# B&R Automation Studio project PrintMark
Automation Studio 4.12.2.93; technology packages: Acp10Arnc0 5.24.1, mapp 5.24.2, mappView 5.24.1

## Configuration Config1

CPU X20CP1584, AutomationRuntime B4.93, Build 4.1.2, Vc V4.72.6

### Task classes (Cpu.sw)
```
Cyclic#1 (cycle 1600 us, tolerance 1600 us):
  BeltCtrl <- SOURCE.BeltCtrl.BeltCtrl.prg  // This task is for controlling the belt conveyor
  CutterCtrl <- SOURCE.CutterCtrl.CutterCtrl.prg  // This task is for controlling the cutter axis
  RegMkCtrl <- SOURCE.RegMark.RegMkCtrl.prg  // This task is for reg mark capture
Cyclic#4 (cycle 99200 us, tolerance 99200 us):
  VisCtrl <- SOURCE.VisCtrl.VisCtrl.prg  // This task if for Hmi task control
  MainCtrl <- SOURCE.MainCtrl.MainCtrl.prg
DataObjects: Acp10sys
NcDataObjects: acp10etxen <- acp10etxen.dob, gBeltAxisa <- gBeltAxisobj.gBeltAxisa.dob, gBeltAxisi <- gBeltAxisobj.gBeltAxisi.dob, gCutAxisa <- gCutAxisobj.gCutAxisa.dob, gCutAxisi <- gCutAxisobj.gCutAxisi.dob
Binaries: FWRules, TCData, udbdef, TCLang, arsvcreg, mvLoader, acp10cfg, Acp10map, iomap, arconfig, asfw, ashwac, sysconf, User, Role, ashwd, BeltConfig, TC, CutConfig, PrintAlarm, PrintCom
Libraries: Acp10man, Acp10par, NcGlobal, Acp10_MC, sys_lib, brsystem, runtime, MpPackML, MpBase, astime, MpAxis, MpCom, standard, MpAlarmX, MpServer, MC_RegMa, fileio, powerlnk, arssl, asbrstr, asieccon, dataobj, aruser
```

### Hardware
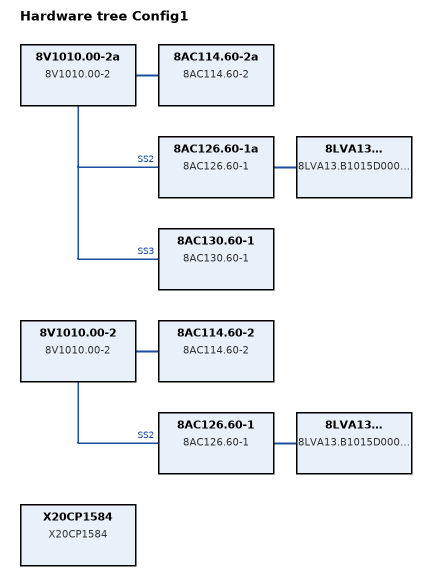
```
8AC114.60-2 : 8AC114.60-2 v1.0.0.8  [SS -> 8V1010.00-2.SS1; PLK1 -> X20CP1584.IF3 (NodeNumber=1) [Cable Type=PowerlinkCable, Length=10, Version=1.0.0.3]; PLK2 -> 8AC114.60-2a.PLK1 (NodeNumber=1) [Cable Type=PowerlinkCable, Length=10, Version=1.0.0.3]]
8AC114.60-2a : 8AC114.60-2 v1.0.0.8  [SS -> 8V1010.00-2a.SS1; PLK1 -> 8AC114.60-2.PLK2 (NodeNumber=2) [Cable Type=PowerlinkCable, Length=10, Version=1.0.0.3]]
8AC126.60-1 : 8AC126.60-1 v2.2.0.0  [SS -> 8V1010.00-2.SS2]
8AC126.60-1a : 8AC126.60-1 v2.2.0.0  [SS -> 8V1010.00-2a.SS2]
8AC130.60-1 : 8AC130.60-1 v2.2.0.0  [SS -> 8V1010.00-2a.SS3]
8LVA13.B1015D000-0 : 8LVA13.B1015D000-0 v2.2.0.3  [EC -> 8AC126.60-1.EC; MT -> 8V1010.00-2.MT1]
8LVA13.B1015D000-0a : 8LVA13.B1015D000-0 v2.2.0.3  [EC -> 8AC126.60-1a.EC; MT -> 8V1010.00-2a.MT1]
8V1010.00-2 : 8V1010.00-2 v2.2.0.0
  MotionTP = Acp10Arnc0
  SinglePhaseOperation = on
  BothEndSwitchesAreNormallyOpen_r1 = on
  QuickStopIsNormallyOpen_r1 = on
8V1010.00-2a : 8V1010.00-2 v2.2.0.0
  MotionTP = Acp10Arnc0
  SinglePhaseOperation = on
  AxisIsPeriodic_r1 = on
  Period_r1 = 3600
  BothEndSwitchesAreNormallyOpen_r1 = on
  QuickStopIsNormallyOpen_r1 = on
X20CP1584 : X20CP1584 v1.10.0.0
  Connector IF2:
    ActivateDevice = 1
    Mode = Manual
    InternetAddress = 192.168.0.11
    SubnetMask = 255.255.255.0
    ActivateSnmp = 2
  Connector IF3:
    CycleTime = 1600
  ConfigurationID = PrintMark_Config1
  TimerDeviceType = EPLX2X
  TimerDevice = X20CP1584.IF3
  TaskClassIdleTime = 1600
  Cyclic1Duration = 1600
  Cyclic1Tolerance = 1600
  Cyclic2Duration = 19200
  Cyclic2Tolerance = 19200
  Cyclic3Duration = 49600
  Cyclic3Tolerance = 49600
  Cyclic4Duration = 99200
  Cyclic4Tolerance = 99200
  Cyclic6Duration = 499200
  Cyclic6Tolerance = 499200
  Cyclic8Duration = 9600
  FileDevice1
  FileDeviceName1 = USER
  FileDevicePath1 = USER_PATH
  FileDevice2
  FileDeviceName2 = Print
  FileDevicePath2 = C:\
  FtpUser1
  FtpUsername1 = printmark
  FtpUserPassword1 = J40jtcY6ygfeMe3/XVHLOVhutVx6SKtWgX0BANt4QHs=
  FtpUserSalt1 = 8YC+oSMn
  FTPAccessRight1 = 0
  FTPdevice1 = ALL
  ActivateOpcUa = 1
  OpcUaInformationModels_PV_Version = 1
```

### Acp10cfg.ncc - X20CP1584/Motion/Acp10cfg.ncc
```
NcConfiguration (Version=5.24.1, NcSwId=Acp10)
  ACP10CF1_typ:
    cnt_nettrc_rec_drive = 1500
    bufsize_trace_upload = 1200
    tc_nc_man_task = Cyclic #1
    glob_pv_as_ncobject = Yes
    ncsys_dl_broadcast = Yes
    ncsys_dl_acp_reset = Yes
    safemc_log_err_to_ax = Yes
    network_init:
      ncsw_init_execute = Yes
      automatic_execute = Yes
      node_nr_warning = Yes
      net_err_before_ncact = Yes
    nettrc:
      enter_parsecrec = Yes
      enter_ncaction = Yes
      save_ring_startidx = Yes
    cam_prof_download:
      cam_dat_dl_parallel = No
      tc_cam_dl_parallel = Task class for NC Manager task
    plk_if[0]:
      if_name = IF3
      tc_CycDat_PLCopen = Task class for NC Manager task
      mc_broadcast_extdat = No
```

### Acp10map.ncm - X20CP1584/Motion/Acp10map.ncm
```
NcMapping (NcSwId=Acp10, DisabledNodesAreHidden=False)
  NcObject 8V1010.00-2_ncV_AXIS1 (ModuleId=8V1010.00-2, Type=ncV_AXIS, Channel=1, Disabled=TRUE, ModuleDisabled=FALSE)
  NcObject 8V1010.00-2a_ncV_AXIS1 (ModuleId=8V1010.00-2a, Type=ncV_AXIS, Channel=1, Disabled=TRUE, ModuleDisabled=FALSE)
  NcObject gBeltAxis (ModuleId=8V1010.00-2, Type=ncAXIS, Channel=1, AcoposSimulation=Off, InitParameter=gBeltAxisi, AcoposParameter=gBeltAxisa, Disabled=FALSE, ModuleDisabled=FALSE)  // This axis is for Belt conveyor
  NcObject gCutAxis (ModuleId=8V1010.00-2a, Type=ncAXIS, Channel=1, AcoposSimulation=Off, InitParameter=gCutAxisi, AcoposParameter=gCutAxisa, AdditionalData=PLCopen_ModPos="3600,1" , Disabled=FALSE, ModuleDisabled=FALSE)  // This axis is for Cutter unit
```

### BeltConfig.mpaxisbasic - X20CP1584/Motion/BeltConfig.mpaxisbasic
```
Element gMl_BeltAxis (Type=mpaxisbasic)
  Alarms = MpAlarmX
```

### CutConfig.mpaxisbasic - X20CP1584/Motion/CutConfig.mpaxisbasic
```
Element gMl_CutAxis (Type=mpaxisbasic)
  Alarms = MpAlarmX
```

### PrintAlarm.mpalarmxcore - X20CP1584/mappServices/PrintAlarm.mpalarmxcore
```
Element gMl_PrintAlarm (Type=mpalarmxcore)
  mapp.AlarmX.Core.Configuration:
    [0]:
      Name = Estop
      Message = Machine E-Stop is pressed
      Behavior = PersistentAlarm
    [1]:
      Name = BeltTempError
      Message = Belt conveyor motor temperature is high
      Behavior = PersistentAlarm
    [2]:
      Name = CutterTempError
      Message = Cutter conveyor motor is temperature is high
      Behavior = PersistentAlarm
    [3]:
      Name = CuttingZone
      Message = Cutter is in cutting zone please move it manually
      Behavior = PersistentAlarm
```

### PrintCom.mpcomgroup - X20CP1584/mappServices/PrintCom.mpcomgroup
```
Element gMl_PrintChildGroup (Type=mpcomgroup)
  Linking:
    Subnodes:
      0 = gMl_BeltAxis
      1 = gMl_CutAxis
      2 = gMl_PrintAlarm
  Alarms = MpAlarmX
Element gMl_PrintParentGroup (Type=mpcomgroup)
  Linking:
    Subnodes:
      0 = gMl_PrintChildGroup
  Alarms = MpAlarmX
```

### PrintData.mpdatarecorder - X20CP1584/mappServices/PrintData.mpdatarecorder
```
Element gMl_PrintDataRecorder (Type=mpdatarecorder)
```

### PrintPack.mppackmlcore - X20CP1584/mappServices/PrintPack.mppackmlcore
```
Element gMl_PrintPackML (Type=mppackmlcore)
  Modes:
    Mode[1]:
      ModeID = 1
      Name = Automatic
    Mode[2]:
      ModeID = 2
      Name = Mode[3]
```

## Logical view

Binary libraries used (declarations not repeated): operator, runtime, astime, AsIecCon, Acp10man, Acp10par, NcGlobal, Acp10_MC, sys_lib, brsystem, MpPackML, MpBase, MpAxis, standard, MpAlarmX, MpServer, MC_RegMa 5.24.1

### Global.typ - Global data types
```iecst
(*Structure for axis control*)

TYPE
	AxisBasicIn_type : 	STRUCT  (*Axis Basic inputs structure type*)
		ErrorReset : BOOL; (*Resets function block errors*) (* *) (*#PAR#;*)
		Parameters : MpAxisBasicParType; (*Function block parameters*) (* *) (*#PAR#;*)
		Update : BOOL; (*Updates the parameters*) (* *) (*#PAR#;*)
		Power : BOOL; (*Level-sensitive command for turning an axis on/off. In the event of an error, a new rising edge is required to restart the axis*) (* *) (*#CMD#;*)
		Home : BOOL; (*Command for homing the axis*) (* *) (*#CMD#;*)
		MoveVelocity : BOOL; (*Starts a constant movement with a defined velocity*) (* *) (*#CMD#;*)
		MoveAbsolute : BOOL; (*Starts an absolute movement*) (* *) (*#CMD#;*)
		MoveAdditive : BOOL; (*Starts a relative movement*) (* *) (*#CMD#;*)
		Stop : BOOL; (*Stops the axis*) (* *) (*#CMD#;*)
		JogPositive : BOOL; (*Movement in the positive direction. Stops automatically at the software limit position*) (* *) (*#CMD#OPT#;*)
		JogNegative : BOOL; (*Movement in the negative direction. Stops automatically at the software limit position*) (* *) (*#CMD#OPT#;*)
		Autotune : BOOL; (*Starts autotuning*) (* *) (*#CMD#OPT#;*)
		Simulate : BOOL; (*Enables motor simulation*) (* *) (*#CMD#OPT#;*)
		TorqueLimit : BOOL; (*Enables torque limiting*) (* *) (*#CMD#OPT#;*)
		ReleaseBrake : BOOL; (*Locks or unlocks the holding brake (only when the axis is switched off)*) (* *) (*#CMD#OPT#;*)
	END_STRUCT;
	AxisBasicOut_type : 	STRUCT  (*Axis Basic outputs structure type*)
		Active : BOOL; (*Indicates whether the function block is active*) (* *) (*#PAR#;*)
		Error : BOOL; (*Indicates that the function block is in an error state or a command was not executed correctly*) (* *) (*#PAR#;*)
		StatusID : DINT; (*Status information about the function block*) (* *) (*#PAR#;*)
		UpdateDone : BOOL; (*Parameter update completed*) (* *) (*#PAR#;*)
		Position : LREAL; (*Current position of the axis [units]*) (* *) (*#CYC#;*)
		Velocity : REAL; (*Current position of the axis [units/s]*) (* *) (*#CYC#;*)
		CommandBusy : BOOL; (*Function block currently executing command*) (* *) (*#CMD#OPT#;*)
		CommandAborted : BOOL; (*Function block interrupted while executing a command*) (* *) (*#CMD#OPT#;*)
		PowerOn : BOOL; (*Switches on the axis*) (* *) (*#CMD#;*)
		IsHomed : BOOL; (*Homes the axis*) (* *) (*#CMD#;*)
		InVelocity : BOOL; (*Axis running with defined velocity*) (* *) (*#CMD#;*)
		InPosition : BOOL; (*Axis reached the desired position*) (* *) (*#CMD#;*)
		MoveActive : BOOL; (*Movement active*) (* *) (*#CMD#;*)
		Stopped : BOOL; (*Axis stopped*) (* *) (*#CMD#;*)
		TuningDone : BOOL; (*Autotuning completed successfully*) (* *) (*#CMD#OPT#;*)
		Simulation : BOOL; (*Motor simulation active*) (* *) (*#CMD#OPT#;*)
		TorqueLimited : BOOL; (*Torque limiting function active*) (* *) (*#CMD#OPT#;*)
		BrakeReleased : BOOL; (*Holding brake manually released*) (* *) (*#CMD#OPT#;*)
		Info : MpAxisBasicInfoType; (*Additional information about the component*) (* *) (*#CMD#;*)
	END_STRUCT;
	AxisBasic_type : 	STRUCT  (*Axis Basic structure type*)
		In : AxisBasicIn_type;
		Out : AxisBasicOut_type;
	END_STRUCT;
	AxisCamSeqIn_type : 	STRUCT  (*Axis cam sequencing input structure type*)
		ErrorReset : BOOL; (*Resets function block errors*) (* *) (*#PAR#;*)
		Parameters : MpAxisCamSequencerParType; (*Function block parameters*) (* *) (*#PAR#;*)
		Update : BOOL; (*Update command for the parameters*) (* *) (*#PAR#;*)
		Signal1 : BOOL; (*Sets the signal for the sequencer on a rising edge and resets the signal on a falling edge*) (* *) (*#CMD#;*)
		Signal2 : BOOL; (*Sets the signal for the sequencer on a rising edge and resets the signal on a falling edge*) (* *) (*#CMD#;*)
		Signal3 : BOOL; (*Sets the signal for the sequencer on a rising edge and resets the signal on a falling edge*) (* *) (*#CMD#OPT#;*)
		Signal4 : BOOL; (*Sets the signal for the sequencer on a rising edge and resets the signal on a falling edge*) (* *) (*#CMD#OPT#;*)
		StartSequence : BOOL; (*Starts the cam sequencer*) (* *) (*#CMD#OPT#;*)
		Continue : BOOL; (*To continue the cam sequencer if standby was active*)
		EndSequence : BOOL; (*Stops the cam sequencer*)
	END_STRUCT;
	AxisCamSeqOut_type : 	STRUCT  (*Axis cam sequencing output structure type*)
		Active : BOOL; (*Indicates whether the function block is active*) (* *) (*#PAR#;*)
		Error : BOOL; (*Indicates that the function block is in an error state or a command was not executed correctly*) (* *) (*#PAR#;*)
		StatusID : DINT; (*Status information about the function block*) (* *) (*#PAR#;*)
		UpdateDone : BOOL; (*Parameter update completed*) (* *) (*#PAR#;*)
		ActualStateIndex : USINT; (*Index of the current state. *) (* *) (*#CMD#OPT#;*)
		ActualStateCamIndex : UINT; (*Index of curve being used in the current state*) (* *) (*#CMD#OPT#;*)
		StandBy : BOOL; (*The cam sequencer can be started using the continue command*) (* *) (*#CMD#;*)
		InCompensation : BOOL; (*Axis currently performing a compensating movement*) (* *) (*#CMD#;*)
		InSync : BOOL; (*Slave synchronous with the master*) (* *) (*#CMD#OPT#;*)
		Info : MpAxisCamSequencerInfoType; (*Additional information about the component*) (* *) (*#CMD#;*)
	END_STRUCT;
	AxisCamSeq_type : 	STRUCT  (*Axis cam sequencing type*)
		In : AxisCamSeqIn_type;
		Out : AxisCamSeqOut_type;
	END_STRUCT;
END_TYPE

(*Structure for machine control*)

TYPE
	PrintCmd_Typ : 	STRUCT
		Start : BOOL; (*Start command for the machine*)
		Stop : BOOL; (*Stop command for the machine*)
		JogPositive : BOOL; (*Jog positive command for the machine*)
		JogNegative : BOOL; (*Jog Negative command for the machine*)
		ErrorAck : BOOL; (*Error acknowledge command for the machine*)
		Estop : BOOL; (*E-Stop for the machine*)
	END_STRUCT;
	PrintPara_Typ : 	STRUCT
		MachineSpeed : REAL; (*Machine speed parameter*)
		New_Member : USINT;
	END_STRUCT;
	PrintStatus_Typ : 	STRUCT  (*Structure for showing the status of the machine*)
		machineStatus : STRING[80]; (*For displaying status of the machine*)
		powerOnHome : BOOL; (*For checking homing*)
	END_STRUCT;
	PrintIn_Typ : 	STRUCT  (*Structure for Inputs of the machine*)
		New_Member : USINT;
	END_STRUCT;
	PrintOut_Typ : 	STRUCT  (*Structure for outputs of the machine*)
		New_Member : USINT;
	END_STRUCT;
	PrintIO_Typ : 	STRUCT  (*Structure for IO's of the machine*)
		Input : PrintIn_Typ;
		Output : PrintOut_Typ;
	END_STRUCT;
	PrintCtrl_Typ : 	STRUCT  (*Structure of controlling the machine operation*)
		Cmd : PrintCmd_Typ; (*Machine command type variable*)
		Para : PrintPara_Typ; (*Machine parameters type variable*)
		Status : PrintStatus_Typ; (*Machine status type variable*)
		IO : PrintIO_Typ; (*Machine IO type variable*)
	END_STRUCT;
END_TYPE
```

### Global.var - Global variables
```iecst
(*Global variable for axis control*)
VAR
	gAx_BeltConveyor : AxisBasic_type; (*Master type varibale*)
	gAx_Cutter : AxisBasic_type; (*Slave basic type variable*)
	gAx_CutterCam : AxisCamSeq_type := (0); (*Slave cam sequencing type variable*)
	gBeltAxis : ACP10AXIS_typ; (*This axis is for controlling the Belt axis*)
	gCutAxis : ACP10AXIS_typ; (*This axis is for controlling the Cutter axis*)
	gRegAdvancePara : MC_BR_ADV_RM2_REF; (*MC_BR_RegMarkCapture002 Adavnced parameter type variable*)
	gRegConfigPara : MC_BR_CFG_RM2_REF; (*MC_BR_RegMarkCapture002 Configuration parameter type variable*)
END_VAR
(*Global variable for machine control*)
VAR
	gPrintMark : PrintCtrl_Typ; (*Variable for Print mark machine control*)
	gPrintMarkHMI : PrintCtrHMIl_Typ; (*Variable for Print mark visualization control*)
END_VAR
```


### Package Logical/gBeltAxisobj - gBeltAxisobj

### Data object Logical/gBeltAxisobj/gBeltAxisa (Apt)

#### gBeltAxisa.apt
```
AcoposParameterTable:
  Root Parameters:
    484 = 111 (Name=MA1_CYCLIC_SEND)  // Network coupling: Parameter ID of send data master1
```

### Data object Logical/gBeltAxisobj/gBeltAxisi (Ax)

#### gBeltAxisi.ax
```
InitParameter (Version=5.24.1, NcSwId=ACP10)
  ACP10AXIS_typ:
    dig_in:
      level:
        reference = ncACTIV_HI + ncFORCE
        pos_hw_end = ncACTIV_HI
        neg_hw_end = ncACTIV_HI
        trigger1 = ncACTIV_HI
        trigger2 = ncACTIV_HI
    encoder_if:
      parameter:
        count_dir = ncSTANDARD
        scaling:
          load:
            units = 1600
            rev_motor = 1
    limit:
      parameter:
        v_pos = 120000.0
        v_neg = 120000.0
        a1_pos = 1.2E+07
        a2_pos = 1.2E+07
        a1_neg = 1.2E+07
        a2_neg = 1.2E+07
        t_jolt = 0.01
        t_in_pos = 0.0
        pos_sw_end = 8388607
        neg_sw_end = -8388608
        ds_warning = 180.0
        ds_stop = 360.0
        a_stop = 1.0E+30
        dv_stop = 0.0
        dv_stop_mode = ncOFF
    controller:
      mode = ncPOSITION
      position:
        kv = 456.0
        tn = 0.0
        t_predict = 0.0024
        t_total = 0.0024
        p_max = 1.0E+30
        i_max = 0.0
      speed:
        kv = 0.6
        tn = 0.0
        t_filter = 0.0
        isq_filter1:
          type = ncOFF
          a0 = 0.0
          a1 = 0.0
          b0 = 0.0
          b1 = 0.0
          b2 = 0.0
          c0_par_id = 0
          c1_par_id = 0
        isq_filter2:
          type = ncOFF
          a0 = 0.0
          a1 = 0.0
          b0 = 0.0
          b1 = 0.0
          b2 = 0.0
          c0_par_id = 0
          c1_par_id = 0
        isq_filter3:
          type = ncOFF
          a0 = 0.0
          a1 = 0.0
          b0 = 0.0
          b1 = 0.0
          b2 = 0.0
          c0_par_id = 0
          c1_par_id = 0
      uf:
        type = ncLINEAR + ncCORRECTION
        auto_config = ncMOTOR_PAR
        u0 = 0.0
        un = 0.0
        fn = 50.0
        k_f_slip = 0.0
      ff:
        mode = ncSTANDARD
        torque_load = 0.0
        torque_pos = 0.0
        torque_neg = 0.0
        kv_torque = 0.0
        inertia = 0.0
        t_filter_a = 0.0
      fb:
        mode = ncSTANDARD
        speed_mix_ratio = 0.0
        speed_kv = 0.0
      model:
        mass1:
          inertia = 0.0
          viscous_friction = 0.0
        mass2:
          inertia = 0.0
          viscous_friction = 0.0
          stiffness = 0.0
          damping = 0.0
    move:
      stop:
        parameter[0]:
          decel_ramp = ncA_LIMIT
          controller = ncON
        parameter[1]:
          decel_ramp = ncA_LIMIT
          controller = ncON
        parameter[2]:
          decel_ramp = ncA_LIMIT
          controller = ncON
        parameter[3]:
          decel_ramp = ncA_LIMIT
          controller = ncON
        quickstop:
          decel_ramp = ncA_LIMIT
          t_jolt = 0.0
        drive_error:
          decel_ramp = ncA_LIMIT
      homing:
        parameter:
          s = 0
          v_switch = 5000.0
          v_trigger = 500.0
          a = 50000.0
          mode = ncDIRECT
          edge_sw = ncPOSITIVE
          start_dir = ncPOSITIVE
          trigg_dir = ncPOSITIVE
          ref_pulse = ncOFF
          fix_dir = ncOFF
          tr_s_block = 0.0
          torque_lim = 0.0
          ds_block = 0.0
          ds_stop = 0.0
      basis:
        parameter:
          v_pos = 5000.0
          v_neg = 5000.0
          a1_pos = 50000.0
          a2_pos = 50000.0
          a1_neg = 50000.0
          a2_neg = 50000.0
    message:
      text:
        parameter:
          format = ncBREAK + ncZERO
          columns = 80
          data_modul = acp10etxen
```

### Package Logical/gCutAxisobj - gCutAxisobj

### Data object Logical/gCutAxisobj/gCutAxisa (Apt)

#### gCutAxisa.apt - Parameter table
```
AcoposParameterTable:
  Root Parameters:
    593 = 1,484 (Name=CONFIG_MA1_CYCLIC_POS)  // Network coupling: Configure station to receive on MA1_CYCLIC_POS
    CAMCON:
      777 = 10752 (Name=FUNCTION_BLOCK_CREATE)  // Function block: Create a FB instance
      10752 = 0 (Name=CAMCON_MODE+0)  // FB0 CAMCON Mode
      10760 = 542 (Name=CAMCON_IN_PARID+0)  // FB0 CAMCON Parameter ID of input
      10864 (Name=CAMCON_EV_PARID+0, Disabled=TRUE)  // FB0 CAMCON Parameter ID start event
      10768 = 0 (Name=CAMCON_S_START+0)  // FB0 CAMCON Start position
      10776 = 700 (Name=CAMCON_S_IV+0)  // FB0 CAMCON Interval
      10784 (Name=CAMCON_T_DELAY_ON+0, Unit=s, Disabled=TRUE)  // FB0 CAMCON Delay time to switch output ON
      10792 (Name=CAMCON_T_DELAY_OFF+0, Unit=s, Disabled=TRUE)  // FB0 CAMCON Delay time to switch output OFF
      10800 (Name=CAMCON_T1_DELAY+0, Unit=s, Disabled=TRUE)  // FB0 CAMCON Switch delay: Filter time constant
      10808 (Name=CAMCON_HYSTERESIS+0, Disabled=TRUE)  // FB0 CAMCON Hysteresis window
      10816 = 1 (Name=CAMCON_MAX_CAM+0, Disabled=FALSE)  // FB0 CAMCON Maximum number of cams
      10824 = 1 (Name=CAMCON_CAM_INDEX+0)  // FB0 CAMCON Index of parameter record for one cam
      10832 = 600 (Name=CAMCON_CAM_S1+0)  // FB0 CAMCON Start position of cam within interval
      10840 = 690 (Name=CAMCON_CAM_S2+0)  // FB0 CAMCON End position of cam within interval
      10848 = 0 (Name=CAMCON_VALUE+0)  // FB0 CAMCON Output value
      10752 = 1 (Name=CAMCON_MODE+0)  // FB0 CAMCON Mode
```

### Data object Logical/gCutAxisobj/gCutAxisi (Ax)

#### gCutAxisi.ax - Init table
```
InitParameter (Version=5.24.1, NcSwId=ACP10)
  ACP10AXIS_typ:
    dig_in:
      level:
        reference = ncACTIV_HI
        pos_hw_end = ncACTIV_HI
        neg_hw_end = ncACTIV_HI
        trigger1 = ncACTIV_HI
        trigger2 = ncACTIV_HI
    encoder_if:
      parameter:
        count_dir = ncINVERSE
        scaling:
          load:
            units = 3600
            rev_motor = 1
    limit:
      parameter:
        v_pos = 120000.0
        v_neg = 120000.0
        a1_pos = 1.2E+07
        a2_pos = 1.2E+07
        a1_neg = 1.2E+07
        a2_neg = 1.2E+07
        t_jolt = 0.01
        t_in_pos = 0.0
        pos_sw_end = 2000000000
        neg_sw_end = -2000000000
        ds_warning = 180.0
        ds_stop = 360.0
        a_stop = 1.0E+30
        dv_stop = 0.0
        dv_stop_mode = ncOFF
    controller:
      mode = ncPOSITION
      position:
        kv = 311.0
        tn = 0.0
        t_predict = 0.0024
        t_total = 0.0024
        p_max = 1.0E+30
        i_max = 0.0
      speed:
        kv = 0.7
        tn = 0.0
        t_filter = 0.0
        isq_filter1:
          type = ncOFF
          a0 = 0.0
          a1 = 0.0
          b0 = 0.0
          b1 = 0.0
          b2 = 0.0
          c0_par_id = 0
          c1_par_id = 0
        isq_filter2:
          type = ncOFF
          a0 = 0.0
          a1 = 0.0
          b0 = 0.0
          b1 = 0.0
          b2 = 0.0
          c0_par_id = 0
          c1_par_id = 0
        isq_filter3:
          type = ncOFF
          a0 = 0.0
          a1 = 0.0
          b0 = 0.0
          b1 = 0.0
          b2 = 0.0
          c0_par_id = 0
          c1_par_id = 0
      uf:
        type = ncLINEAR + ncCORRECTION
        auto_config = ncMOTOR_PAR
        u0 = 0.0
        un = 0.0
        fn = 50.0
        k_f_slip = 0.0
      ff:
        mode = ncSTANDARD
        torque_load = 0.0
        torque_pos = 0.0
        torque_neg = 0.0
        kv_torque = 0.0
        inertia = 0.0
        t_filter_a = 0.0
      fb:
        mode = ncSTANDARD
        speed_mix_ratio = 0.0
        speed_kv = 0.0
      model:
        mass1:
          inertia = 0.0
          viscous_friction = 0.0
        mass2:
          inertia = 0.0
          viscous_friction = 0.0
          stiffness = 0.0
          damping = 0.0
    move:
      stop:
        parameter[0]:
          decel_ramp = ncA_LIMIT
          controller = ncON
        parameter[1]:
          decel_ramp = ncA_LIMIT
          controller = ncON
        parameter[2]:
          decel_ramp = ncA_LIMIT
          controller = ncON
        parameter[3]:
          decel_ramp = ncA_LIMIT
          controller = ncON
        quickstop:
          decel_ramp = ncA_LIMIT
          t_jolt = 0.0
        drive_error:
          decel_ramp = ncA_LIMIT
      homing:
        parameter:
          s = 0
          v_switch = 5000.0
          v_trigger = 500.0
          a = 50000.0
          mode = ncDIRECT
          edge_sw = ncPOSITIVE
          start_dir = ncPOSITIVE
          trigg_dir = ncPOSITIVE
          ref_pulse = ncON
          fix_dir = ncOFF
          tr_s_block = 0.0
          torque_lim = 0.0
          ds_block = 0.0
          ds_stop = 0.0
      basis:
        parameter:
          v_pos = 5000.0
          v_neg = 5000.0
          a1_pos = 50000.0
          a2_pos = 50000.0
          a1_neg = 50000.0
          a2_neg = 50000.0
    message:
      text:
        parameter:
          format = ncBREAK
          columns = 80
          data_modul = acp10etxen
```

### Package Logical/SOURCE - Source file for logical control

### Program Logical/SOURCE/MainCtrl/MainCtrl (IEC)

#### Main.st - Init, cyclic, exit code
```iecst
PROGRAM _INIT
	//Local pointer method to access other modules
	beltConvStatus := PV_xgetadr(ADR('BeltCtrl:beltCtrl'),ADR(beltConvAddress),ADR(beltConvSize));
	cutterStatus := PV_xgetadr(ADR('CutterCtrl:cutCtrl'),ADR(cutterAddress),ADR(cutterSize));
END_PROGRAM

PROGRAM _CYCLIC
	//For Accessing Variables of Other Modules
	pBeltConveyorCtrl ACCESS beltConvAddress;
	pCutterCtrl ACCESS cutterAddress;

	//Calling Auto mode action file
	Automatic;
END_PROGRAM

PROGRAM _EXIT
	(* Insert code here *)

END_PROGRAM
```

#### Types.typ - Local data types
```iecst
TYPE
	enAutoMode :
		( (*Enumeraton for auto mode operation*)
		CLEARING,
		HELD,
		IDLE,
		STARTING,
		EXECUTE,
		STOPPING,
		ABORTED
		);
END_TYPE
```

#### Variables.var - Local variables
```iecst
(*Variable for Auto mode*)
VAR
	startRising : BOOL;
	startFound : BOOL;
	stopPressed : BOOL;
	eStopPressed : BOOL;
	emergencyFault : BOOL;
	errorAckRising : BOOL;
	errorAckFound : BOOL;
	enAutoStep : enAutoMode;
	machineReady : BOOL;
END_VAR
(*Constants*)
VAR CONSTANT
	K_ACC_FACTOR : UINT := 10;
	K_DEC_FACTOR : UINT := 10;
	CAM_SEQUENCING : BOOL := TRUE; (*CAM Sequencing Mode*)
	K_ZERO : REAL := 0.0; (*Constant for zero value*)
	K_STOP_PHASE : REAL := 360.0; (*Constant for stop in phase*)
END_VAR
(*Local Pointer method variables for accessing other modules*)
VAR
	beltConvStatus : UINT; (*Return Variable for pvxgetaddress of Belt Conv module*)
	beltConvAddress : UDINT; (*Pointer address for Belt Conv control*)
	beltConvSize : UDINT; (*Size of belt conveyor pointer variable*)
	pBeltConveyorCtrl : REFERENCE TO BeltCtrl_Typ; (*Pointer variable for accessing Belt conveyor module*)
	cutterStatus : UINT; (*Return Variable for pvxgetaddress of Cutter module*)
	cutterAddress : UDINT; (*Pointer address for Cutter control*)
	cutterSize : UDINT; (*Size of cutter pointer variable*)
	pCutterCtrl : REFERENCE TO CutterCtrl_Typ; (*Pointer variable for accessing Cutter module*)
END_VAR
```

#### Automatic.st
```iecst
ACTION Automatic:

	//Basic input parameters for the machine
	//Start command
	startRising := (gPrintMark.Cmd.Start = TRUE) AND (startFound = FALSE);
	startFound  := (gPrintMark.Cmd.Start = TRUE);
	//Error Reset
	errorAckRising := (gPrintMark.Cmd.ErrorAck = TRUE) AND (errorAckFound = FALSE);
	errorAckFound  := (gPrintMark.Cmd.ErrorAck = TRUE);
	gAx_BeltConveyor.In.ErrorReset := errorAckRising;
	gAx_Cutter.In.ErrorReset := errorAckRising;
	gAx_CutterCam.In.ErrorReset := errorAckRising;
	//Updating the FB's
	gAx_BeltConveyor.In.Update := FALSE;
	gAx_Cutter.In.Update := FALSE;
	gAx_CutterCam.In.Update := FALSE;
	//Speed parameters
	gAx_BeltConveyor.In.Parameters.Velocity := gPrintMark.Para.MachineSpeed;
	gAx_BeltConveyor.In.Parameters.Acceleration := gPrintMark.Para.MachineSpeed * K_ACC_FACTOR ;
	gAx_BeltConveyor.In.Parameters.Deceleration := gPrintMark.Para.MachineSpeed * K_DEC_FACTOR;

	//Stop command for the machine
	IF (gAx_BeltConveyor.Out.MoveActive = TRUE) AND
		(gAx_BeltConveyor.Out.Info.PLCopenState = mpAXIS_CONTINUOUS_MOTION) AND
		(gPrintMark.Cmd.Stop = TRUE) THEN
		stopPressed := TRUE;
	END_IF

	//Estop and emergency conditions for the machine
	IF (gPrintMark.Cmd.Estop = TRUE) THEN
		eStopPressed := TRUE;
	ELSIF (gPrintMark.Cmd.Estop = TRUE) AND (errorAckRising = TRUE) THEN
		eStopPressed := FALSE;
	END_IF

	IF (gAx_BeltConveyor.Out.StatusID <> 0) OR (gAx_BeltConveyor.Out.Error = TRUE) OR
		(gAx_Cutter.Out.StatusID <> 0) OR (gAx_Cutter.Out.Error = TRUE) OR
		(gAx_CutterCam.Out.StatusID <> 0) OR (eStopPressed = TRUE) THEN
		emergencyFault := TRUE;
	ELSE
		emergencyFault := FALSE;
	END_IF

	//State machine for the Auto mode
	CASE enAutoStep OF
		CLEARING:	//For checking any error in the machine
			gPrintMark.Status.machineStatus := 'Machine is Healthy';
			machineReady := FALSE;
			IF (gAx_BeltConveyor.Out.Active = TRUE) AND
				(gAx_Cutter.Out.Active = TRUE) AND
				(gAx_CutterCam.Out.Active = TRUE) AND
				(gAx_BeltConveyor.Out.Info.BootState = mpAXIS_BLP_DONE) AND
				(gAx_Cutter.Out.Info.BootState = mpAXIS_BLP_DONE) THEN
				gAx_BeltConveyor.In.Power := TRUE;
				gAx_Cutter.In.Power := TRUE;
				enAutoStep := HELD;
			END_IF

		HELD:	//Giving Power ON and Homing command for the axis
			gPrintMark.Status.machineStatus := 'Axis Power ON and Homing';
			IF (gAx_BeltConveyor.Out.PowerOn = TRUE) AND
				(gAx_Cutter.Out.PowerOn = TRUE) THEN
				IF (gPrintMark.Status.powerOnHome = FALSE) THEN
					pBeltConveyorCtrl.Cmd.bHome := TRUE;
					pCutterCtrl.Cmd.bHome := TRUE;
				END_IF
			END_IF
			IF (gAx_BeltConveyor.Out.IsHomed = TRUE) AND
				((gAx_Cutter.Out.IsHomed = TRUE)OR(gAx_Cutter.Out.Position = 0)) THEN
				gPrintMark.Status.powerOnHome := TRUE;
				pBeltConveyorCtrl.Cmd.bHome := FALSE;
				pCutterCtrl.Cmd.bHome := FALSE;
				enAutoStep := IDLE;
			END_IF

		IDLE:	//Waiting for Start Command
			gPrintMark.Status.machineStatus := 'Machine Waiting for Start Command';
			machineReady := TRUE;
			IF (startRising = TRUE) AND
				(gPrintMark.Cmd.Stop = FALSE) AND
				(gPrintMark.Cmd.Estop = FALSE) THEN
				IF (CAM_SEQUENCING = TRUE) THEN
					gAx_CutterCam.In.StartSequence := TRUE;
					gAx_CutterCam.In.EndSequence := FALSE;
				END_IF
				enAutoStep := STARTING;
			END_IF

		STARTING:	//Starting the CAM Sequence
			IF (CAM_SEQUENCING <> TRUE) THEN
				gAx_CutterCam.In.StartSequence := FALSE;
				gAx_CutterCam.In.EndSequence := FALSE;
			END_IF
			gAx_BeltConveyor.In.MoveVelocity := TRUE;
			enAutoStep := EXECUTE;

		EXECUTE: //Starting the Master Axis
			gPrintMark.Status.machineStatus := 'Machine is in Motion';
			IF (stopPressed = TRUE) THEN
				gAx_BeltConveyor.In.Stop := TRUE;
				gAx_BeltConveyor.In.Parameters.Stop.StopInPhase := TRUE;
				gAx_BeltConveyor.In.Parameters.Stop.Phase := K_STOP_PHASE;
				gAx_BeltConveyor.In.Parameters.Stop.Deceleration := gPrintMark.Para.MachineSpeed * K_DEC_FACTOR;
				enAutoStep := STOPPING;
			END_IF

		STOPPING:	//Stopping the master axis
			gPrintMark.Status.machineStatus := 'Machine Stopping in Phase';
			IF (gAx_BeltConveyor.Out.Stopped = TRUE) THEN
				gAx_BeltConveyor.In.MoveVelocity := FALSE;
				gAx_BeltConveyor.In.Stop := FALSE;
				stopPressed := FALSE;
				enAutoStep := ABORTED;
			END_IF

		ABORTED:	//Error Acknowledgement
			gPrintMark.Status.machineStatus := 'Machine is in Error';
			IF (gAx_BeltConveyor.Out.Stopped = TRUE) OR
				(gAx_BeltConveyor.Out.Info.PLCopenState = mpAXIS_ERRORSTOP) OR
				(gAx_BeltConveyor.Out.Info.PLCopenState = mpAXIS_DISABLED) THEN
				gAx_BeltConveyor.In.Stop := FALSE;
			END_IF

			IF (gAx_BeltConveyor.Out.PowerOn = FALSE) THEN
				gAx_BeltConveyor.In.Power := FALSE;
			END_IF

			IF (gAx_Cutter.Out.PowerOn = FALSE) THEN
				gAx_Cutter.In.Power := FALSE;
			END_IF

			IF (gAx_Cutter.Out.Stopped = TRUE) OR
				(gAx_Cutter.Out.Info.PLCopenState = mpAXIS_ERRORSTOP) OR
				(gAx_Cutter.Out.Info.PLCopenState = mpAXIS_DISABLED) THEN
				gAx_CutterCam.In.StartSequence := FALSE;
				gAx_Cutter.In.Stop  := FALSE;
			END_IF

			IF (emergencyFault = FALSE) AND
				((gAx_BeltConveyor.Out.Info.PLCopenState = mpAXIS_DISABLED) OR (gAx_BeltConveyor.Out.Info.PLCopenState = mpAXIS_STANDSTILL)) AND
				((gAx_Cutter.Out.Info.PLCopenState = mpAXIS_DISABLED) OR (gAx_Cutter.Out.Info.PLCopenState = mpAXIS_STANDSTILL)) THEN
				enAutoStep := CLEARING;
			END_IF
	END_CASE;

	//Actions to be performed in case of emergency
	IF (emergencyFault = TRUE) AND (enAutoStep < CLEARING) THEN
		enAutoStep := ABORTED;
		gAx_BeltConveyor.In.Stop := TRUE;
		gAx_BeltConveyor.In.Parameters.Stop.StopInPhase  := FALSE;
		gAx_BeltConveyor.In.Parameters.Stop.Deceleration := K_ZERO;

		gAx_Cutter.In.Stop := TRUE;
		gAx_Cutter.In.Parameters.Stop.StopInPhase  := FALSE;
		gAx_Cutter.In.Parameters.Stop.Deceleration := K_ZERO;

	END_IF
	IF (emergencyFault = TRUE) THEN
		machineReady := FALSE;
		gAx_BeltConveyor.In.MoveVelocity := FALSE;
		gAx_BeltConveyor.Out.IsHomed := FALSE;
		gAx_Cutter.Out.IsHomed := FALSE;
		gAx_BeltConveyor.In.Power := FALSE;
		gAx_Cutter.In.Power := FALSE;
		gPrintMark.Status.powerOnHome := FALSE;
	END_IF

END_ACTION
```

#### PrintAlarm.st - not listed in the package file held
```iecst
ACTION PrintAlarm:

	//Alarms for temperature
	IF(gAx_BeltConveyor.Out.Info.CyclicRead.MotorTemperature.Value >= K_MAX_TEMP)THEN
		Alarm[1] := TRUE;
	ELSE
		Alarm[1] := FALSE;
	END_IF;
	IF(gAx_Cutter.Out.Info.CyclicRead.MotorTemperature.Value >= K_MAX_TEMP)THEN
		Alarm[2] := TRUE;
	ELSE
		Alarm[2] := FALSE;
	END_IF;

	//Alarm for homing in cutting zone
	IF(gPrintMark.Status.cuttingZone = TRUE)THEN
		Alarm[3] := TRUE;
	ELSE
		Alarm[3] := FALSE;
	END_IF;

END_ACTION
```

### Program Logical/SOURCE/BeltCtrl/BeltCtrl (IEC)

#### Main.st - Init, cyclic, exit code
```iecst
(*|ŻŻŻŻŻŻŻŻŻŻŻŻŻŻŻŻŻŻŻŻŻŻŻŻŻŻŻŻŻŻŻŻŻŻŻŻŻŻŻŻŻŻŻŻŻŻŻŻŻŻŻŻŻŻŻŻŻŻŻŻŻŻŻŻŻŻŻŻŻŻŻŻŻŻ|*)
(*| Copyright      :- B&R Industrial Automation GmbH                         |*)
(*| Contact Person :-   kuma1p                                      		 |*)
(*|——————————————————————————————————————————————————————————————————————————|*)
(*| System       :-  Machine Name                                            |*)
(*| Task Name    :-  BeltCtrl.st                                             |*)
(*| Auther Name  :-   kuma1p                                       			 |*)
(*| Created Date :-May 8, 2024/1:04 AM                                       |*)
(*| AS Version   :-  AS 4.12.2.93                                            |*)
(*|——————————————————————————————————————————————————————————————————————————|*)
(*| Description  :-  This task is for Belt conveyor control                  |*)
(*|                                                                          |*)
(*|——————————————————————————————————————————————————————————————————————————|*)
(*| Version :-         V 0.0                      kuma1p                     |*)
(*|Changes Made :-  Axio IO Action file and Homing                           |*)
(*| Version :-         V 0.1                      kuma1p                     |*)
(*|Changes Made :-  Manual operation action file                             |*)
(*|——————————————————————————————————————————————————————————————————————————|*)
PROGRAM _INIT
	beltCtrl.Para.homeVelocity := K_HOME_VEL_INIT;
END_PROGRAM

PROGRAM _CYCLIC

	//Calling Belt Axis IO mapping file
	AxisIOMap;

	//Calling Belt Axis Homing file
	IF(gPrintMark.Cmd.ManualMode = TRUE)THEN
		beltCtrl.Cmd.bHome := gPrintMarkHMI.Cmd.bBeltHome;
	END_IF;
	Homing;

	//Calling Belt Axis manual operation
	IF(gPrintMark.Cmd.ManualMode = TRUE)THEN
		beltCtrl.Para.jogSpeed := gPrintMarkHMI.Para.beltJogSpeed;
		beltCtrl.Cmd.bJogPositive := gPrintMarkHMI.Cmd.bBeltJogPositive;
		beltCtrl.Cmd.bJogNegative := gPrintMarkHMI.Cmd.bBeltJogNegative;
		Manual;
	END_IF;

END_PROGRAM

PROGRAM _EXIT
	iFb_MpAxisBasic.Enable := FALSE;
	iFb_MpAxisBasic();
END_PROGRAM
```

#### Types.typ - Local data types
```iecst
(*Enumerations*)

TYPE
	enBeltManualMode :
		( (*Enumeration for manual mode movement of Belt axis*)
		IDLE, (*Idle state in manual mode*)
		STARTING, (*Starting state in manual mode*)
		EXECUTE, (*Execute state in manual mode*)
		ABORTING (*Aborting state in manual mode*)
		);
	enBeltHomeMode :
		( (*Enumeration for homing of belt axis*)
		HOME_IDLE, (*Idle state in manual mode*)
		HOME_STARTING, (*Starting state in manual mode*)
		HOME_EXECUTE, (*Execute state in manual mode*)
		HOME_STOPPING, (*Stopping state in manual mode*)
		HOME_STOPPED (*Stopped state in manual mode*)
		);
END_TYPE
```

#### Variables.var - Local variables
```iecst
(*MpAxisBasic type variable*)
VAR
	iFb_MpAxisBasic : MpAxisBasic; (*Belt Mp Axis Basic Variable*)
	iFb_MC_BR_SetHardwareInputs : MC_BR_SetHardwareInputs;
END_VAR
(*Enumeration variable*)
VAR
	enBeltManualSteps : enBeltManualMode; (*Enumeration type variable for manual mode*)
	enBeltHomeSteps : enBeltHomeMode; (*Enumeration type variable for homing*)
END_VAR
(*Variable for belt unit control*)
VAR
	beltCtrl : BeltCtrl_Typ; (*Variable of Belt ctrl type*)
	negLimitAbort : BOOL; (*Variable for aborting negative belt jog*)
	prohibitNegJog : BOOL; (*Prohibiting negative jog*)
END_VAR
(*Constants*)
VAR CONSTANT
	K_BELT_ACC_FACTOR : UINT := 10; (*Constant for giving  acceleration*)
	K_BELT_DEC_FACTOR : UINT := 10; (*Constant for giving  decelaration*)
	K_UNIT_PER_REV : UINT := 1600; (*constant for belt axis units per revolution*)
	K_QUARTER : UINT := 4; (*constant for quarter value*)
	K_HALF : UINT := 2; (*constant for half value*)
	K_CORRECTION : UINT := 60; (*constant for homing position correction*)
	K_ZERO : UINT := 0; (*constant for zero value*)
	K_HOME_POS_OFFSET : UINT := 8; (*constant for home offset*)
	K_HOME_VEL_INIT : REAL := 100; (*Homing velocuty *)
	K_JOG_NEG_LIMIT : REAL := 300; (*Negative limit while negative jog*)
	K_PERIOD : UINT := 3600; (*Period of belt axis motion*)
	K_HALF_PERIOD : UINT := 1800; (*Half period of belt axis motion*)
END_VAR
(*FB Types *)
VAR
	iFb_RtrigBeltJog : R_TRIG; (*R_Trig FB type variable*)
END_VAR
```

#### AxisIOMap.st - Belt Axis Mapping
```iecst
ACTION AxisIOMap:

	//Belt Axis Basic inputs
	iFb_MpAxisBasic.MpLink       := ADR(gMl_BeltAxis);
	iFb_MpAxisBasic.Enable       := TRUE;
	iFb_MpAxisBasic.ErrorReset   := gAx_BeltConveyor.In.ErrorReset;
	iFb_MpAxisBasic.Parameters   := ADR(gAx_BeltConveyor.In.Parameters);
	iFb_MpAxisBasic.Update       := gAx_BeltConveyor.In.Update;
	iFb_MpAxisBasic.Axis         := ADR(gBeltAxis);
	iFb_MpAxisBasic.Power        := gAx_BeltConveyor.In.Power;
	iFb_MpAxisBasic.Home         := gAx_BeltConveyor.In.Home;
	iFb_MpAxisBasic.MoveVelocity := gAx_BeltConveyor.In.MoveVelocity;
	iFb_MpAxisBasic.MoveAbsolute := gAx_BeltConveyor.In.MoveAbsolute;
	iFb_MpAxisBasic.MoveAdditive := gAx_BeltConveyor.In.MoveAdditive;
	iFb_MpAxisBasic.Stop         := gAx_BeltConveyor.In.Stop;
	iFb_MpAxisBasic.JogPositive  := gAx_BeltConveyor.In.JogPositive;
	iFb_MpAxisBasic.JogNegative  := gAx_BeltConveyor.In.JogNegative;
	iFb_MpAxisBasic.Autotune     := gAx_BeltConveyor.In.Autotune;
	iFb_MpAxisBasic.Simulate     := gAx_BeltConveyor.In.Simulate;
	iFb_MpAxisBasic.TorqueLimit  := gAx_BeltConveyor.In.TorqueLimit;
	iFb_MpAxisBasic.ReleaseBrake := gAx_BeltConveyor.In.ReleaseBrake;
	iFb_MpAxisBasic();

	//Belt Axis Basic outputs
	gAx_BeltConveyor.Out.Active         := iFb_MpAxisBasic.Active;
	gAx_BeltConveyor.Out.Error          := iFb_MpAxisBasic.Error;
	gAx_BeltConveyor.Out.StatusID       := iFb_MpAxisBasic.StatusID;
	gAx_BeltConveyor.Out.UpdateDone     := iFb_MpAxisBasic.UpdateDone;
	gAx_BeltConveyor.Out.Position       := iFb_MpAxisBasic.Position;
	gAx_BeltConveyor.Out.Velocity       := iFb_MpAxisBasic.Velocity;
	gAx_BeltConveyor.Out.CommandBusy    := iFb_MpAxisBasic.CommandBusy;
	gAx_BeltConveyor.Out.CommandAborted := iFb_MpAxisBasic.CommandAborted;
	gAx_BeltConveyor.Out.PowerOn        := iFb_MpAxisBasic.PowerOn;
	gAx_BeltConveyor.Out.IsHomed        := iFb_MpAxisBasic.IsHomed;
	gAx_BeltConveyor.Out.InVelocity     := iFb_MpAxisBasic.InVelocity;
	gAx_BeltConveyor.Out.InPosition     := iFb_MpAxisBasic.InPosition;
	gAx_BeltConveyor.Out.MoveActive     := iFb_MpAxisBasic.MoveActive;
	gAx_BeltConveyor.Out.Stopped        := iFb_MpAxisBasic.Stopped;
	gAx_BeltConveyor.Out.TuningDone     := iFb_MpAxisBasic.TuningDone;
	gAx_BeltConveyor.Out.Simulation     := iFb_MpAxisBasic.Simulation;
	gAx_BeltConveyor.Out.TorqueLimited  := iFb_MpAxisBasic.TorqueLimited;
	gAx_BeltConveyor.Out.BrakeReleased  := iFb_MpAxisBasic.BrakeReleased;
	gAx_BeltConveyor.Out.Info           := iFb_MpAxisBasic.Info;

	//For homing of Belt conveyor
	iFb_MC_BR_SetHardwareInputs.Enable := TRUE;
	iFb_MC_BR_SetHardwareInputs.Axis := ADR(gBeltAxis);
	iFb_MC_BR_SetHardwareInputs.HomeSwitch := gAx_Cutter.Out.Info.DigitalInputsStatus.Trigger1;
	iFb_MC_BR_SetHardwareInputs();

END_ACTION
```

#### Manual.st - Action file for manual belt operation
```iecst
ACTION Manual:

	//Updating jog speed for the belt axis
	gAx_BeltConveyor.In.Parameters.Jog.Velocity := beltCtrl.Para.jogSpeed;
	gAx_BeltConveyor.In.Parameters.Jog.Acceleration := beltCtrl.Para.jogSpeed * K_BELT_ACC_FACTOR;
	gAx_BeltConveyor.In.Parameters.Jog.Deceleration := beltCtrl.Para.jogSpeed * K_BELT_DEC_FACTOR;
	IF(gAx_BeltConveyor.In.Parameters.Jog.Velocity <> beltCtrl.Para.jogSpeed)THEN
		gAx_BeltConveyor.In.Update := TRUE;
		IF(gAx_BeltConveyor.Out.UpdateDone = TRUE)THEN
			gAx_BeltConveyor.In.Update := FALSE;
		END_IF;
	END_IF;

	//Case for manual operation of belt axis
	CASE enBeltManualSteps OF
		IDLE: //Idle state for the state machine
			IF((gAx_BeltConveyor.Out.PowerOn = TRUE) AND (gAx_BeltConveyor.Out.Error = FALSE))THEN
				enBeltManualSteps := STARTING;
			END_IF;

		STARTING: //Starting parameters for the state machine;
			enBeltManualSteps := EXECUTE;

		EXECUTE: //Executing jog positive and negative
			gAx_BeltConveyor.In.Parameters.Jog.LowerLimit := K_ZERO;
			gAx_BeltConveyor.In.Parameters.Jog.UpperLimit := K_ZERO;
			IF((gAx_BeltConveyor.In.Parameters.Jog.LowerLimit <> K_ZERO) OR
				(gAx_BeltConveyor.In.Parameters.Jog.UpperLimit <> K_ZERO))THEN
				gAx_BeltConveyor.In.Update := TRUE;
				IF(gAx_BeltConveyor.Out.UpdateDone = TRUE)THEN
					gAx_BeltConveyor.In.Update := FALSE;
				END_IF;
			END_IF;
			IF(beltCtrl.Cmd.bJogPositive = TRUE)THEN
				prohibitNegJog := FALSE;
				gAx_BeltConveyor.In.JogPositive := TRUE;
			ELSE
				gAx_BeltConveyor.In.JogPositive := FALSE;
			END_IF;
			IF((beltCtrl.Cmd.bJogNegative = TRUE) AND (prohibitNegJog = FALSE))THEN
				IF(gAx_Cutter.Out.Info.DigitalInputsStatus.Trigger1 = FALSE)THEN
					gAx_BeltConveyor.In.JogNegative := TRUE;
					negLimitAbort := FALSE;
				ELSE
					negLimitAbort := TRUE;
					enBeltManualSteps := ABORTING;
				END_IF;
			ELSE
				gAx_BeltConveyor.In.JogNegative := FALSE;
			END_IF;
			IF((gAx_BeltConveyor.Out.PowerOn = FALSE) OR (gAx_BeltConveyor.Out.Error = TRUE))THEN
				enBeltManualSteps := IDLE;
			END_IF;

		ABORTING: //Aborting the jogging in case of negative limit reached
			IF(iFb_RtrigBeltJog.Q)THEN
				IF((gAx_BeltConveyor.Out.Position > K_ZERO) AND
					(gAx_BeltConveyor.Out.Position < (K_HALF_PERIOD+K_JOG_NEG_LIMIT)))THEN
					gAx_BeltConveyor.In.Parameters.Jog.LowerLimit := gAx_BeltConveyor.Out.Position - K_JOG_NEG_LIMIT;
					gAx_BeltConveyor.In.Parameters.Jog.UpperLimit := ((K_PERIOD)-(gAx_BeltConveyor.Out.Position - K_JOG_NEG_LIMIT));
				ELSIF((gAx_BeltConveyor.Out.Position < K_PERIOD) AND
					(gAx_BeltConveyor.Out.Position >= (K_HALF_PERIOD+K_JOG_NEG_LIMIT)))THEN
					gAx_BeltConveyor.In.Parameters.Jog.UpperLimit := K_PERIOD;
					gAx_BeltConveyor.In.Parameters.Jog.LowerLimit := (gAx_BeltConveyor.Out.Position - K_JOG_NEG_LIMIT);
				END_IF;
			END_IF;
			IF((gAx_BeltConveyor.In.Parameters.Jog.LowerLimit <> K_ZERO) OR
				(gAx_BeltConveyor.In.Parameters.Jog.UpperLimit <> K_ZERO))THEN
				gAx_BeltConveyor.In.Update := TRUE;
				IF(gAx_BeltConveyor.Out.UpdateDone = TRUE)THEN
					gAx_BeltConveyor.In.Update := FALSE;
				END_IF;
			END_IF;
			IF(gAx_BeltConveyor.Out.Velocity = K_ZERO)THEN
				prohibitNegJog := TRUE;
				negLimitAbort := FALSE;
				gAx_BeltConveyor.In.JogNegative := FALSE;
				enBeltManualSteps := EXECUTE;
			END_IF;
			IF((gAx_BeltConveyor.Out.PowerOn = FALSE) OR (gAx_BeltConveyor.Out.Error = TRUE))THEN
				enBeltManualSteps := IDLE;
			END_IF;
			IF(beltCtrl.Cmd.bJogNegative = FALSE)THEN
				gAx_BeltConveyor.In.JogNegative := FALSE;
			END_IF;

	END_CASE;

	//Calling R_TRIG FB
	iFb_RtrigBeltJog(CLK := negLimitAbort);

END_ACTION
```

#### Homing.st - Action file for Homing operation
```iecst
ACTION Homing:

	CASE enBeltHomeSteps OF
		HOME_IDLE: //Idle state for homing
			IF((gAx_BeltConveyor.Out.PowerOn = TRUE) AND (gAx_BeltConveyor.Out.Error = FALSE))THEN
				enBeltHomeSteps := HOME_STARTING;
			END_IF;

		HOME_STARTING: //Starting command for the homing
			gAx_BeltConveyor.In.Parameters.Home.Mode := mpAXIS_HOME_MODE_ABS_SWITCH;
			gAx_BeltConveyor.In.Parameters.Home.HomingVelocity := beltCtrl.Para.homeVelocity;
			gAx_BeltConveyor.In.Parameters.Home.Acceleration := beltCtrl.Para.homeVelocity * K_BELT_ACC_FACTOR;
			enBeltHomeSteps := HOME_EXECUTE;

		HOME_EXECUTE: //Executing homing for the axis
			IF(beltCtrl.Cmd.bHome = TRUE)THEN
				gAx_BeltConveyor.In.Home := TRUE;
				enBeltHomeSteps := HOME_STOPPING;
			END_IF;

		HOME_STOPPING: //Homing is being stopped
			IF(gAx_BeltConveyor.Out.IsHomed = TRUE)THEN
				enBeltHomeSteps := HOME_STOPPED;
			END_IF;

		HOME_STOPPED: //Homing is stopped
			gAx_BeltConveyor.In.Home := FALSE;
			IF(gAx_BeltConveyor.Out.Velocity = K_ZERO)THEN
				enBeltHomeSteps := HOME_IDLE;
			END_IF;
	END_CASE;

END_ACTION
```

### BeltTyp.typ - not listed in the package file held
```iecst
(*Belt conveyor section controlling structure*)

TYPE
	BeltCmd_Typ : 	STRUCT  (*Structure for giving command to belt conveyor section*)
		bStart : BOOL; (*Start command*)
		bStop : BOOL; (*Stop command*)
		bHome : BOOL; (*Home command*)
		bJogPositive : BOOL; (*Positive jog command*)
		bJogNegative : BOOL; (*Negative jog command*)
	END_STRUCT;
	BeltPara_Typ : 	STRUCT  (*Structure for giving the parameters to belt conveyor section*)
		jogSpeed : REAL; (*For giving jog speed to the belt unit*)
		jogUpperLimit : REAL; (*For giving jog upper limit to the belt unit*)
		jogLowerLimit : REAL; (*For giving jog lower limit to the belt unit*)
		homeVelocity : REAL; (*Homing velocity*)
		homeAccel : REAL; (*Homing acceleration*)
		homeDecel : REAL; (*Homing deceleration*)
	END_STRUCT;
	BeltStatus_Typ : 	STRUCT  (*Strcuture for showing the status of the belt conveyor section*)
		New_Member : USINT;
	END_STRUCT;
	BeltCtrl_Typ : 	STRUCT  (*Structure for controlling the belt conveyor section*)
		Cmd : BeltCmd_Typ; (*Giving command to the belt conveyor section*)
		Para : BeltPara_Typ; (*Giving parameters to the belt conveyor section*)
		Status : BeltStatus_Typ; (*Getting status of the belt conveyor section*)
	END_STRUCT;
END_TYPE
```

### Program Logical/SOURCE/CutterCtrl/CutterCtrl (IEC)

#### Main.st - Init, cyclic, exit code
```iecst
PROGRAM _INIT
	cutCtrl.Para.homeVelocity := K_HOME_VEL_INIT;
	cutCtrl.Para.homePositiveTol := ((K_UNIT_PER_REV)/K_HALF)-(K_HOME_POS_TOL);
	cutCtrl.Para.homeNegativeTol := ((K_UNIT_PER_REV)/K_HALF)+(K_HOME_NEG_TOL);
END_PROGRAM

PROGRAM _CYCLIC

	//Calling Cutter Axis IO mapping file
	AxisIOMap;

	//Calling Cutter Axis Homing Command
	HomePos;

	//Homing Operation after finding homing position
	cutCtrl.Cmd.bHome := gPrintMarkHMI.Cmd.bCutterHome;
	IF(cutCtrl.Status.bHomePosFound = TRUE)THEN
		Homing;
	END_IF;

	//Manual command for Cutter axis
	Manual;
	cutCtrl.Para.jogSpeed := gPrintMarkHMI.Para.cutterJogSpeed;
	cutCtrl.Cmd.bJogPositive := gPrintMarkHMI.Cmd.bCutterJogPositive;
	cutCtrl.Cmd.bJogNegative := gPrintMarkHMI.Cmd.bCutterJogNegative;

	//Cam Automat
	Printcam;

END_PROGRAM

PROGRAM _EXIT
	iFb_MpAxisBasic.Enable := FALSE;
	iFb_MpAxisBasic();

END_PROGRAM
```

#### Types.typ - Local data types
```iecst
(*Enumerations*)

TYPE
	enCutterHomeMode :
		( (*Enumeration for cutter homing state machine*)
		HOME_IDLE, (*Idle state in manual mode*)
		HOME_STARTING, (*Starting state in manual mode*)
		HOME_EXECUTE, (*Execute state in manual mode*)
		HOME_STOPPING, (*Stopping state in manual mode*)
		HOME_STOPPED (*Stopped state in manual mode*)
		);
	enCutterManualMode :
		( (*Enumeration for cutter manual mode state machine*)
		IDLE, (*Idle state in manual mode*)
		STARTING, (*Starting state in manual mode*)
		EXECUTE (*Execute state in manual mode*)
		);
END_TYPE
```

#### Variables.var - Local variables
```iecst
(*MpAxisBasic type variable*)
VAR
	iFb_MpAxisBasic : MpAxisBasic; (*Cutter Mp Axis Basic Variable*)
	iFb_MpAxisCaming : MpAxisCamSequencer; (*MpAxis Cam Sequencer variable*)
END_VAR
(*Enumeration variable*)
VAR
	enCutterHomeSteps : enCutterHomeMode; (*Enumeration type variable for homing*)
	enCutterManualSteps : enCutterManualMode; (*Enumeration type variable for manual operation*)
END_VAR
(*Cutting unit ctrl*)
VAR
	cutCtrl : CutterCtrl_Typ; (*Variable of Cutter control type*)
	cutHomePostion : REAL; (*Home postition for cutter axis*)
END_VAR
(*Constants*)
VAR CONSTANT
	K_CUT_ACC_FACTOR : UINT := 10; (*constant for cutting axis acceleration*)
	K_CUT_DEC_FACTOR : UINT := 10; (*constant for cutting axis deceleration*)
	K_UNIT_PER_REV : UINT := 3600; (*constant for cut axis units per revolution*)
	K_QUARTER : UINT := 4; (*constant for quarter value*)
	K_HALF : UINT := 2; (*constant for half value*)
	K_CUTTER_ANGLE : UINT := 360; (*constant for cutter disc angle*)
	K_CORRECTION : UINT := 60; (*constant for homing position correction*)
	K_ZERO : UINT := 0; (*constant for zero value*)
	K_HOME_POS_TOL : UINT := 200; (*constant for positive tolerance for homing*)
	K_HOME_NEG_TOL : UINT := 200; (*constant for negative tolerance for homing*)
	K_HOME_POS_OFFSET : UINT := 8; (*constant for home offset*)
	K_HOME_LOW_RANGE : UINT := 420; (*Lower range for finding home position*)
	K_HOME_UP_RANGE : UINT := 1140; (*Upper range for finding home position*)
	K_HOME_VEL_INIT : REAL := 100; (*Homing velocuty *)
	K_ONE : UINT := 1; (*Constant value 1*)
END_VAR
```

#### AxisIOMap.st
```iecst
ACTION AxisIOMap:

	//Cutter Axis Basic Input
	iFb_MpAxisBasic.MpLink       := ADR(gMl_CutAxis);
	iFb_MpAxisBasic.Enable       := TRUE;
	iFb_MpAxisBasic.ErrorReset   := gAx_Cutter.In.ErrorReset;
	iFb_MpAxisBasic.Parameters   := ADR(gAx_Cutter.In.Parameters);
	iFb_MpAxisBasic.Update       := gAx_Cutter.In.Update;
	iFb_MpAxisBasic.Axis         := ADR(gCutAxis);
	iFb_MpAxisBasic.Power        := gAx_Cutter.In.Power;
	iFb_MpAxisBasic.Home         := gAx_Cutter.In.Home;
	iFb_MpAxisBasic.MoveVelocity := gAx_Cutter.In.MoveVelocity;
	iFb_MpAxisBasic.MoveAbsolute := gAx_Cutter.In.MoveAbsolute;
	iFb_MpAxisBasic.MoveAdditive := gAx_Cutter.In.MoveAdditive;
	iFb_MpAxisBasic.Stop         := gAx_Cutter.In.Stop;
	iFb_MpAxisBasic.JogPositive  := gAx_Cutter.In.JogPositive;
	iFb_MpAxisBasic.JogNegative  := gAx_Cutter.In.JogNegative;
	iFb_MpAxisBasic.Autotune     := gAx_Cutter.In.Autotune;
	iFb_MpAxisBasic.Simulate     := gAx_Cutter.In.Simulate;
	iFb_MpAxisBasic.TorqueLimit  := gAx_Cutter.In.TorqueLimit;
	iFb_MpAxisBasic.ReleaseBrake := gAx_Cutter.In.ReleaseBrake;
	iFb_MpAxisBasic();

	//Cutter axis Basic Output
	gAx_Cutter.Out.Active         := iFb_MpAxisBasic.Active;
	gAx_Cutter.Out.Error          := iFb_MpAxisBasic.Error;
	gAx_Cutter.Out.StatusID       := iFb_MpAxisBasic.StatusID;
	gAx_Cutter.Out.UpdateDone     := iFb_MpAxisBasic.UpdateDone;
	gAx_Cutter.Out.Position       := iFb_MpAxisBasic.Position;
	gAx_Cutter.Out.Velocity       := iFb_MpAxisBasic.Velocity;
	gAx_Cutter.Out.CommandBusy    := iFb_MpAxisBasic.CommandBusy;
	gAx_Cutter.Out.CommandAborted := iFb_MpAxisBasic.CommandAborted;
	gAx_Cutter.Out.PowerOn        := iFb_MpAxisBasic.PowerOn;
	gAx_Cutter.Out.IsHomed        := iFb_MpAxisBasic.IsHomed;
	gAx_Cutter.Out.InVelocity     := iFb_MpAxisBasic.InVelocity;
	gAx_Cutter.Out.InPosition     := iFb_MpAxisBasic.InPosition;
	gAx_Cutter.Out.MoveActive     := iFb_MpAxisBasic.MoveActive;
	gAx_Cutter.Out.Stopped        := iFb_MpAxisBasic.Stopped;
	gAx_Cutter.Out.TuningDone     := iFb_MpAxisBasic.TuningDone;
	gAx_Cutter.Out.Simulation     := iFb_MpAxisBasic.Simulation;
	gAx_Cutter.Out.TorqueLimited  := iFb_MpAxisBasic.TorqueLimited;
	gAx_Cutter.Out.BrakeReleased  := iFb_MpAxisBasic.BrakeReleased;
	gAx_Cutter.Out.Info           := iFb_MpAxisBasic.Info;

	//Cam Axis basic input parameters
	iFb_MpAxisCaming.MpLink       := ADR(gMl_CutAxis);
	iFb_MpAxisCaming.Enable       := TRUE;
	iFb_MpAxisCaming.ErrorReset   := gAx_CutterCam.In.ErrorReset;
	iFb_MpAxisCaming.Parameters   := ADR(gAx_CutterCam.In.Parameters);
	iFb_MpAxisCaming.Update       := gAx_CutterCam.In.Update;
	iFb_MpAxisCaming.MpLinkMaster := ADR(gMl_BeltAxis);
	iFb_MpAxisCaming.Signal1      := gAx_CutterCam.In.Signal1;
	iFb_MpAxisCaming.Signal2      := gAx_CutterCam.In.Signal2;
	iFb_MpAxisCaming.Signal3      := gAx_CutterCam.In.Signal3;
	iFb_MpAxisCaming.Signal4      := gAx_CutterCam.In.Signal4;
	iFb_MpAxisCaming.StartSequence:= gAx_CutterCam.In.StartSequence;
	iFb_MpAxisCaming.Continue     := gAx_CutterCam.In.Continue;
	iFb_MpAxisCaming.EndSequence  := gAx_CutterCam.In.EndSequence;

	//Cam Axis basic output parameters
	gAx_CutterCam.Out.InSync := iFb_MpAxisCaming.InSync;
	gAx_CutterCam.Out.Error := iFb_MpAxisCaming.Error;

	//Calling Cam FB
	iFb_MpAxisCaming();

END_ACTION
```

#### HomePos.st - Homing action file
```iecst
ACTION HomePos:

	CASE enCutterHomeSteps OF
		HOME_IDLE: //Idle state for homing
			IF((gAx_Cutter.Out.PowerOn = TRUE) AND (gAx_Cutter.Out.Error = FALSE)
				AND(cutCtrl.Status.bHomePosFound = FALSE))THEN
				enCutterHomeSteps := HOME_STARTING;
			END_IF;

		HOME_STARTING: //Starting command for the homing
			gAx_Cutter.In.Parameters.Home.Mode := mcHOME_DIRECT;
			gAx_Cutter.In.Parameters.Home.ReferencePulse := mpAXIS_HOME_OPTION_ON;
			gAx_Cutter.In.Parameters.Home.HomingVelocity := cutCtrl.Para.homeVelocity;
			gAx_Cutter.In.Parameters.Home.Acceleration := cutCtrl.Para.homeVelocity * K_CUT_ACC_FACTOR;
			IF((gAx_Cutter.Out.Position < K_HOME_LOW_RANGE))THEN
					gPrintMark.Status.cuttingZone := FALSE;
				gAx_Cutter.In.Parameters.Home.HomingDirection := mpAXIS_HOME_DIR_NEGATIVE;
			ELSIF((gAx_Cutter.Out.Position > K_HOME_UP_RANGE))THEN
					gPrintMark.Status.cuttingZone := FALSE;
				gAx_Cutter.In.Parameters.Home.HomingDirection := mpAXIS_HOME_DIR_POSITIVE;
			ELSIF((gAx_Cutter.Out.Position>K_HOME_LOW_RANGE)AND(gAx_Cutter.Out.Position < K_HOME_UP_RANGE))THEN
				gPrintMark.Status.cuttingZone := TRUE;
				cutCtrl.Cmd.bHome := FALSE;
			END_IF;
			IF(cutCtrl.Cmd.bHome = TRUE)THEN
				gAx_Cutter.In.Home := TRUE;
			END_IF;
			IF((gAx_Cutter.Out.Position < (K_ZERO+K_HOME_POS_OFFSET))
				OR(gAx_Cutter.Out.Position > (K_UNIT_PER_REV-K_HOME_POS_OFFSET)))THEN
				enCutterHomeSteps := HOME_EXECUTE;
			END_IF;

		HOME_EXECUTE: //Executing homing for the axis
			gAx_Cutter.In.Home := FALSE;
			gAx_Cutter.In.Parameters.Velocity := cutCtrl.Para.homeVelocity;
			gAx_Cutter.In.Parameters.Acceleration := cutCtrl.Para.homeVelocity * K_CUT_ACC_FACTOR;
			gAx_Cutter.In.Parameters.Deceleration := cutCtrl.Para.homeVelocity;
			gAx_Cutter.In.Parameters.Home.ReferencePulse := mpAXIS_HOME_OPTION_OFF;
			cutHomePostion := ((K_UNIT_PER_REV/K_QUARTER)-(K_CUTTER_ANGLE/K_HALF))+(K_UNIT_PER_REV/K_HALF)+K_CORRECTION;
			gAx_Cutter.In.Parameters.Position := (cutHomePostion);
			gAx_Cutter.In.Parameters.Direction := mpAXIS_DIR_NEGATIVE;
			gAx_Cutter.In.MoveAbsolute := TRUE;
			IF(gAx_Cutter.Out.Position = cutHomePostion)THEN
				gAx_Cutter.In.MoveAbsolute := FALSE;
				enCutterHomeSteps := HOME_STOPPING;
			END_IF;

		HOME_STOPPING: //Homing is being stopped
			gAx_Cutter.In.Home := TRUE;
			IF(gAx_Cutter.Out.Position = K_ZERO)THEN
				enCutterHomeSteps := HOME_STOPPED;
			END_IF;

		HOME_STOPPED: //Homing is stopped
			gAx_Cutter.In.Home := FALSE;
			cutCtrl.Status.bHomePosFound := TRUE;
			IF(gAx_Cutter.Out.Velocity = K_ZERO)THEN
				enCutterHomeSteps := HOME_IDLE;
			END_IF;
	END_CASE;
END_ACTION
```

#### Homing.st - Homing action file
```iecst
ACTION Homing:
	IF((cutCtrl.Cmd.bHome = TRUE) AND (gPrintMark.Cmd.DualCutterEnable = FALSE))THEN
		gAx_Cutter.In.Parameters.Velocity := cutCtrl.Para.homeVelocity;
		gAx_Cutter.In.Parameters.Acceleration := cutCtrl.Para.homeVelocity * K_CUT_ACC_FACTOR;
		gAx_Cutter.In.Parameters.Deceleration := cutCtrl.Para.homeVelocity;
		IF((gAx_Cutter.Out.Position < cutCtrl.Para.homePositiveTol)AND(gAx_Cutter.Out.Position > K_ZERO))THEN
			gAx_Cutter.In.Parameters.Direction := mpAXIS_DIR_NEGATIVE;
			gAx_Cutter.In.Parameters.Position := K_ZERO + cutCtrl.Para.homeOffset;
			gAx_Cutter.In.MoveAbsolute := TRUE;
			gPrintMark.Status.cuttingZone := FALSE;
		ELSIF((gAx_Cutter.Out.Position > cutCtrl.Para.homeNegativeTol)AND(gAx_Cutter.Out.Position < K_UNIT_PER_REV))THEN
			gAx_Cutter.In.Parameters.Direction := mpAXIS_DIR_POSITIVE;
			gAx_Cutter.In.Parameters.Position := K_ZERO + cutCtrl.Para.homeOffset;
			gAx_Cutter.In.MoveAbsolute := TRUE;
			gPrintMark.Status.cuttingZone := FALSE;
		ELSIF((gAx_Cutter.Out.Position>cutCtrl.Para.homePositiveTol)AND
			(gAx_Cutter.Out.Position<cutCtrl.Para.homeNegativeTol))THEN
			cutCtrl.Cmd.bHome := FALSE;
			gPrintMark.Status.cuttingZone := TRUE;
		END_IF;
	ELSIF((gAx_Cutter.Out.Position = K_ZERO))THEN
		gAx_Cutter.In.MoveAbsolute := FALSE;
		gPrintMark.Status.cuttingZone := FALSE;
	END_IF;

END_ACTION
```

#### Manual.st - Manual cutter operation
```iecst
ACTION Manual:

	//Update logic for speed
	gAx_Cutter.In.Parameters.Jog.Velocity := cutCtrl.Para.jogSpeed;
	gAx_Cutter.In.Parameters.Jog.Acceleration := cutCtrl.Para.jogSpeed * K_CUT_ACC_FACTOR;
	gAx_Cutter.In.Parameters.Jog.Deceleration := cutCtrl.Para.jogSpeed * K_CUT_DEC_FACTOR;
	IF(gAx_Cutter.In.Parameters.Jog.Velocity <> cutCtrl.Para.jogSpeed)THEN
		gAx_Cutter.In.Update := TRUE;
		IF(gAx_Cutter.Out.UpdateDone = TRUE)THEN
			gAx_Cutter.In.Update := FALSE;
		END_IF;
	END_IF;

	//Update logic for limits
	gAx_Cutter.In.Parameters.Jog.LowerLimit := cutCtrl.Para.jogLowerLimit;
	gAx_Cutter.In.Parameters.Jog.UpperLimit := 	cutCtrl.Para.jogUpperLimit;
	IF((gAx_Cutter.In.Parameters.Jog.LowerLimit <> cutCtrl.Para.jogLowerLimit) OR
		(gAx_Cutter.In.Parameters.Jog.UpperLimit <> cutCtrl.Para.jogUpperLimit))THEN
		gAx_Cutter.In.Update := TRUE;
		IF(gAx_Cutter.Out.UpdateDone = TRUE)THEN
			gAx_Cutter.In.Update := FALSE;
		END_IF;
	END_IF;

	//Case for manual operation of belt axis
	CASE enCutterManualSteps OF
		IDLE: //Idle state for the state machine
			IF((gAx_Cutter.Out.PowerOn = TRUE) AND (gAx_Cutter.Out.Error = FALSE))THEN
				enCutterManualSteps := STARTING;
			END_IF;

		STARTING: //Starting parametrs for the state machine;
			gAx_Cutter.In.Parameters.Jog.LowerLimit := K_ZERO;
			gAx_Cutter.In.Parameters.Jog.UpperLimit := K_ZERO;
			IF((gAx_Cutter.In.Parameters.Jog.LowerLimit <> K_ZERO) OR
				(gAx_Cutter.In.Parameters.Jog.UpperLimit <> K_ZERO))THEN
				gAx_Cutter.In.Update := TRUE;
				IF(gAx_Cutter.Out.UpdateDone = TRUE)THEN
					gAx_Cutter.In.Update := FALSE;
				END_IF;
			END_IF;
			enCutterManualSteps := EXECUTE;

		EXECUTE: //Executing jog positive and negative
			IF((cutCtrl.Cmd.bJogPositive = TRUE) AND (gAx_Cutter.Out.Position >= K_ZERO)
				AND (gAx_Cutter.Out.Position <= cutCtrl.Para.homePositiveTol))THEN
				cutCtrl.Para.jogLowerLimit := K_ZERO;
				cutCtrl.Para.jogUpperLimit := cutCtrl.Para.homePositiveTol;
				gAx_Cutter.In.JogPositive := TRUE;
			ELSIF((cutCtrl.Cmd.bJogPositive = TRUE) AND (gAx_Cutter.Out.Position >= cutCtrl.Para.homeNegativeTol)
				AND (gAx_Cutter.Out.Position <= K_UNIT_PER_REV))THEN
				cutCtrl.Para.jogUpperLimit := K_UNIT_PER_REV;
				cutCtrl.Para.jogLowerLimit := cutCtrl.Para.homeNegativeTol;
				gAx_Cutter.In.JogPositive := TRUE;
			ELSIF(cutCtrl.Cmd.bJogPositive = FALSE)THEN
				gAx_Cutter.In.JogPositive := FALSE;
			END_IF;
			IF((cutCtrl.Cmd.bJogNegative = TRUE) AND (gAx_Cutter.Out.Position <= cutCtrl.Para.homePositiveTol)
				AND (gAx_Cutter.Out.Position >= K_ZERO))THEN
				cutCtrl.Para.jogLowerLimit := -(K_ONE) ;
				cutCtrl.Para.jogUpperLimit := K_UNIT_PER_REV;
				gAx_Cutter.In.JogNegative := TRUE;
			ELSIF((cutCtrl.Cmd.bJogNegative = TRUE) AND (gAx_Cutter.Out.Position < K_UNIT_PER_REV)
				AND (gAx_Cutter.Out.Position > cutCtrl.Para.homeNegativeTol))THEN
				cutCtrl.Para.jogLowerLimit := cutCtrl.Para.homeNegativeTol ;
				cutCtrl.Para.jogUpperLimit := K_UNIT_PER_REV;
				gAx_Cutter.In.JogNegative := TRUE;
			ELSIF(cutCtrl.Cmd.bJogNegative = FALSE)THEN
				gAx_Cutter.In.JogNegative := FALSE;
			END_IF;
			IF((gAx_Cutter.Out.PowerOn = FALSE) OR (gAx_Cutter.Out.Error = TRUE))THEN
				enCutterManualSteps := IDLE;
			END_IF;

	END_CASE;

END_ACTION
```

#### PrintCam.st - Caming action file single cutter
```iecst
ACTION Printcam:

	gAx_CutterCam.In.Parameters.Configuration.Master := ADR(gMl_BeltAxis); // Not Mplink Axis Address
	gAx_CutterCam.In.Parameters.Configuration.MasterParID := ACP10PAR_PCTRL_S_ACT;  //ACP10PAR_S_SET_VAX1;
	gAx_CutterCam.In.Parameters.Configuration.MaxMasterVelocity := 120000; //Maximum velocity of the master axis.

	(** STATE 0 Event 1 - 	NOT USED - JUMP TO STATE 1 **)
	gAx_CutterCam.In.Parameters.Configuration.State[0].Event[0].Type := ncST_END; //Trigger
	gAx_CutterCam.In.Parameters.Configuration.State[0].Event[0].Attribute := ncAT_ONCE; //Reaction
	gAx_CutterCam.In.Parameters.Configuration.State[0].Event[0].NextState := 1; //Next State

	(** STATE 1 WAIT FOR TRIGGER **)
	gAx_CutterCam.In.Parameters.Configuration.State[1].CamProfileIndex := 16#FFFE;
	gAx_CutterCam.In.Parameters.Configuration.State[1].MasterFactor := 325; //Slope
	gAx_CutterCam.In.Parameters.Configuration.State[1].SlaveFactor := 360; //Slope
	(** STATE 1 WAIT FOR TRIGGER **)
	gAx_CutterCam.In.Parameters.Configuration.State[1].CompMode := ncONLYCOMP;
	gAx_CutterCam.In.Parameters.Configuration.State[1].MasterCompDistance := 225; //Master Positive movement
	gAx_CutterCam.In.Parameters.Configuration.State[1].SlaveCompDistance := 1620; //Slave Positive movement
	(** STATE 1 Event 1 - WAIT FOR S_START **)
	gAx_CutterCam.In.Parameters.Configuration.State[1].Event[0].Type := ncST_END; //Trigger
	gAx_CutterCam.In.Parameters.Configuration.State[1].Event[0].Attribute := ncST_END; //Reaction
	gAx_CutterCam.In.Parameters.Configuration.State[1].Event[0].NextState := 2; //Next State

	(** STATE 2 Event 1- FORWARD MOVEMENT OF SLAVE **)
	gAx_CutterCam.In.Parameters.Configuration.State[2].CamProfileIndex := 16#FFFF;
	gAx_CutterCam.In.Parameters.Configuration.State[2].MasterFactor := 325; //Master Positive movement
	gAx_CutterCam.In.Parameters.Configuration.State[2].SlaveFactor := 360; //Master Positive movement
	(** STATE 2 Event 1- FORWARD MOVEMENT OF SLAVE **)
	gAx_CutterCam.In.Parameters.Configuration.State[2].Event[0].Type := ncST_END; //Trigger
	gAx_CutterCam.In.Parameters.Configuration.State[2].Event[0].Attribute := ncST_END; //Reaction
	gAx_CutterCam.In.Parameters.Configuration.State[2].Event[0].NextState := 3; //Next State

	(** STATE 3 WAIT FOR TRIGGER **)
	gAx_CutterCam.In.Parameters.Configuration.State[3].CamProfileIndex := 16#FFFE;
	gAx_CutterCam.In.Parameters.Configuration.State[3].MasterFactor := 225; //Slope
	gAx_CutterCam.In.Parameters.Configuration.State[3].SlaveFactor := 1620; //Slope
	(** STATE 3 WAIT FOR TRIGGER **)
	gAx_CutterCam.In.Parameters.Configuration.State[3].CompMode := ncONLYCOMP;
	gAx_CutterCam.In.Parameters.Configuration.State[3].MasterCompDistance := 150; //Master Positive movement
	gAx_CutterCam.In.Parameters.Configuration.State[3].SlaveCompDistance := 1620; //Slave Negative movement
	(** STATE 3 Event 1 - WAIT FOR S_START **)
	gAx_CutterCam.In.Parameters.Configuration.State[3].Event[0].Type := ncST_END; //Trigger
	gAx_CutterCam.In.Parameters.Configuration.State[3].Event[0].Attribute := ncST_END; //Reaction
	gAx_CutterCam.In.Parameters.Configuration.State[3].Event[0].NextState := 1; //Next State

END_ACTION
```

#### Home.st - not listed in the package file held
```iecst
ACTION Home:

	CASE enCutterHomeSteps OF
		HOME_IDLE: //Idle state for homing
			IF((gAx_Cutter.Out.PowerOn = TRUE) AND (gAx_Cutter.Out.Error = FALSE))THEN
				enCutterHomeSteps := HOME_STARTING;
			END_IF;

		HOME_STARTING: //Starting command for the homing
			gAx_Cutter.In.Parameters.Home.Mode := mcHOME_DIRECT;
			gAx_Cutter.In.Parameters.Home.ReferencePulse := mpAXIS_HOME_OPTION_ON;
			gAx_Cutter.In.Parameters.Home.HomingVelocity := cutCtrl.Para.homeVelocity;
			gAx_Cutter.In.Parameters.Home.Acceleration := cutCtrl.Para.homeVelocity * K_CUT_ACC_FACTOR;
			IF(cutCtrl.Cmd.bHomePos = TRUE)THEN
				gAx_Cutter.In.Home := TRUE;
				IF(gAx_Cutter.Out.Position = K_ZERO)THEN
					enCutterHomeSteps := HOME_EXECUTE;
				END_IF;
			END_IF;

		HOME_EXECUTE: //Exexuting homing for the axis
			gAx_Cutter.In.Home := FALSE;
			gAx_Cutter.In.Parameters.Velocity := cutCtrl.Para.homeVelocity;
			gAx_Cutter.In.Parameters.Acceleration := cutCtrl.Para.homeVelocity * K_CUT_ACC_FACTOR;
			gAx_Cutter.In.Parameters.Deceleration := cutCtrl.Para.homeVelocity;
			gAx_Cutter.In.Parameters.Home.ReferencePulse := mpAXIS_HOME_OPTION_OFF;
			cutHomePostion := ((K_UNIT_PER_REV/K_QUARTER)-(K_CUTTER_ANGLE/K_HALF))+(K_UNIT_PER_REV/K_HALF)+K_CORRECTION;
			gAx_Cutter.In.Parameters.Position := (cutHomePostion);
			gAx_Cutter.In.Parameters.Direction := mpAXIS_DIR_NEGATIVE;
			gAx_Cutter.In.MoveAbsolute := TRUE;
			IF(gAx_Cutter.Out.Position = cutHomePostion)THEN
				gAx_Cutter.In.MoveAbsolute := FALSE;
				enCutterHomeSteps := HOME_STOPPING;
			END_IF;

		HOME_STOPPING: //Homing is being stopped
			gAx_Cutter.In.Home := TRUE;
			IF(gAx_Cutter.Out.Position = K_ZERO)THEN
				enCutterHomeSteps := HOME_STOPPED;
			END_IF;

		HOME_STOPPED: //Homing is stopped
			gAx_Cutter.In.Home := FALSE;
			IF(gAx_Cutter.Out.Velocity = K_ZERO)THEN
				enCutterHomeSteps := HOME_IDLE;
			END_IF;
	END_CASE;

END_ACTION
```

### CutTyp.typ
```iecst
(*Cutter section controlling structure*)

TYPE
	CutterCmd_Typ : 	STRUCT  (*Structure for giving command to cutter section*)
		bStart : BOOL; (*Start command*)
		bStop : BOOL; (*Stop command*)
		bHomePos : BOOL; (*Command for finding home position*)
		bHome : BOOL; (*Command for homing of cutter axis*)
		bJogPositive : BOOL; (*Command for cutter jog positive*)
		bJogNegative : BOOL; (*Command for cutter jog negative*)
	END_STRUCT;
	CutterPara_Typ : 	STRUCT  (*Structure for giving the parameters to cutter section*)
		homeVelocity : REAL; (*Homing velocity*)
		homeAccel : REAL; (*Homing acceleration*)
		homeDecel : REAL; (*Homing deceleration*)
		homePositiveTol : UINT; (*Tolerance for homing in positive direction*)
		homeNegativeTol : UINT; (*Tolerance for homing in negative direction*)
		homeOffset : UINT; (*Offset for homing*)
		jogSpeed : REAL; (*Cutter axis jog velocity*)
		jogUpperLimit : REAL; (*Cutter axis jog upper limit*)
		jogLowerLimit : REAL; (*Cutter axis jog lower limit*)
	END_STRUCT;
	CutterStatus_Typ : 	STRUCT  (*Strcuture for showing the status of the cutter section*)
		bHomePosFound : BOOL; (*Status for home position found*)
		bHomingDone : BOOL; (*Status for homing done*)
	END_STRUCT;
	CutterCtrl_Typ : 	STRUCT  (*Structure for controlling the cutter section*)
		Cmd : CutterCmd_Typ; (*Giving command to the cutter section*)
		Para : CutterPara_Typ; (*Giving parameters to the cutter section*)
		Status : CutterStatus_Typ; (*Getting status of the belt cutter section*)
	END_STRUCT;
END_TYPE
```

### Program Logical/SOURCE/RegMark/RegMkCtrl (IEC)

#### Types.typ
```iecst
(*RegMark controlling*)

TYPE
	RegMarkCmd_Typ : 	STRUCT  (*Structure for giving command to print mark section*)
		bStartTrigger : BOOL; (*Start Trigger RegMark*)
		bEnableRegMark : BOOL; (*Enable bit for RegMark*)
	END_STRUCT;
	RegMarkPara_Typ : 	STRUCT  (*Structure for giving the parameters to print mark section*)
		productLength : REAL; (*Product length*)
		regMarkPosition : REAL; (*Registration mark position*)
		regMarkOffset : REAL; (*Registrattion mark offset*)
		distanceToSensor : REAL; (*Distance between two sensors*)
		minWidth : REAL; (*Minimun print mark width*)
		maxWidth : REAL; (*maximum print mark width*)
		negWindow : REAL; (*Print mark negative window*)
		posWindow : REAL; (*Print mark positive window*)
		sensorDelay : DINT; (*Print mark sensor delay*)
		correctionValueLimitNeg : REAL; (*Negative correction value*)
		correctionValueLimitPos : REAL; (*Positive correction value*)
	END_STRUCT;
	RegMarkStatus_Typ : 	STRUCT  (*Strcuture for showing the status of the print mark section*)
		New_Member : USINT;
	END_STRUCT;
	RegMarkCtrl_Typ : 	STRUCT  (*Structure for controlling the cutter section*)
		Cmd : RegMarkCmd_Typ; (*Giving command to the print mark section*)
		Para : RegMarkPara_Typ; (*Giving parameters to the cutter section*)
		Status : RegMarkStatus_Typ; (*Getting status of the print mark section*)
	END_STRUCT;
END_TYPE
```

#### Variables.var
```iecst
(*Reg Mark variables*)
VAR
	MC_BR_RegMarkCapture002_Print : MC_BR_RegMarkCapture002 := (0); (*MC_BR_RegMarkCapture002 FB Type variable*)
END_VAR
(*Variable for regmark controlling*)
VAR
	regMarkCtrl : RegMarkCtrl_Typ; (*Variable for regmark controlling*)
END_VAR
(*Constants*)
VAR CONSTANT
	K_INIT_PROD_LENGTH : REAL := 700; (*Init Product length*)
	K_INIT_REGMRK_POS : REAL := 700; (*Init Registration mark position*)
	K_INIT_REGMRK_OFF : REAL := 10; (*Init Registrattion mark offset*)
	K_INIT_SENS_DIST : REAL := 10; (*Init Distance between two sensors*)
	K_INIT_MIN_WIDTH : REAL := 50; (*Init Minimun print mark width*)
	K_INIT_MAX_WIDTH : REAL := 200; (*Init maximum print mark width*)
	K_INIT_WINDOW_NEG : REAL := 200; (*Init Print mark negative window*)
	K_INIT_WINDOW_POS : REAL := 200; (*Init Print mark positive window*)
	K_INIT_SENS_DEL : DINT := 200; (*Init Print mark sensor delay*)
	K_INIT_CORR_NEG : REAL := 70; (*Init Negative correction value*)
	K_INIT_CORR_POS : REAL := 70; (*Init Positive correction value*)
END_VAR
```

#### Main.st
```iecst
PROGRAM _INIT
//	Init values of the Reg mark capture
	regMarkCtrl.Para.productLength := K_INIT_PROD_LENGTH;
	regMarkCtrl.Para.regMarkPosition := K_INIT_REGMRK_POS;
	regMarkCtrl.Para.regMarkOffset := K_INIT_REGMRK_OFF;
	regMarkCtrl.Para.distanceToSensor := K_INIT_SENS_DIST;
	regMarkCtrl.Para.minWidth := K_INIT_MIN_WIDTH;
	regMarkCtrl.Para.maxWidth := K_INIT_MAX_WIDTH;
	regMarkCtrl.Para.negWindow := K_INIT_WINDOW_NEG;
	regMarkCtrl.Para.posWindow := K_INIT_WINDOW_POS;
	regMarkCtrl.Para.sensorDelay := K_INIT_SENS_DEL;
	regMarkCtrl.Para.correctionValueLimitNeg := K_INIT_CORR_NEG;
	regMarkCtrl.Para.correctionValueLimitPos := K_INIT_CORR_POS;
	regMarkCtrl.Cmd.bStartTrigger := TRUE;
	gRegAdvancePara.CorrectCurrentCycle := TRUE;
END_PROGRAM

PROGRAM _CYCLIC

	//	MC_BR_RegMark Config parameters
	gRegConfigPara.ProductLength := regMarkCtrl.Para.productLength;
	gRegConfigPara.RegMarkPosition := regMarkCtrl.Para.regMarkPosition;
	gRegConfigPara.RegMarkOffset := regMarkCtrl.Para.regMarkOffset;
	gRegConfigPara.DistanceToSensor := regMarkCtrl.Para.distanceToSensor;
	//	MC_BR_RegMark Advance parameters
	gRegAdvancePara.Mode := mcFIRST_RM;
	gRegAdvancePara.EventSourceParID := 0;
	gRegAdvancePara.Edge := ncP_EDGE;//Positive Edge
	gRegAdvancePara.MinWidth := regMarkCtrl.Para.minWidth;//Minimum Width of Hole
	gRegAdvancePara.MaxWidth := regMarkCtrl.Para.maxWidth;//Maximum Width of Hole
	gRegAdvancePara.WindowNeg := regMarkCtrl.Para.negWindow;
	gRegAdvancePara.WindowPos := regMarkCtrl.Para.posWindow;
	gRegAdvancePara.SensorDelay := regMarkCtrl.Para.sensorDelay;
	gRegAdvancePara.CorrectionValueLimitNeg := regMarkCtrl.Para.correctionValueLimitNeg;
	gRegAdvancePara.CorrectionValueLimitPos := regMarkCtrl.Para.correctionValueLimitPos;
	//MC_BR_RegMarkCapture002 Type FB
	MC_BR_RegMarkCapture002_Print.Master := ADR(gAx_BeltConveyor);
	MC_BR_RegMarkCapture002_Print.Axis := ADR(gAx_Cutter);
	MC_BR_RegMarkCapture002_Print.Enable := regMarkCtrl.Cmd.bEnableRegMark;
	MC_BR_RegMarkCapture002_Print.SearchRM := regMarkCtrl.Cmd.bStartTrigger;
	MC_BR_RegMarkCapture002_Print.InitData := regMarkCtrl.Cmd.bStartTrigger;
	MC_BR_RegMarkCapture002_Print.CutPosition := REAL_TO_DINT(gRegConfigPara.ProductLength);
	MC_BR_RegMarkCapture002_Print.Configuration := gRegConfigPara;
	MC_BR_RegMarkCapture002_Print.AdvancedParameters := gRegAdvancePara;
	MC_BR_RegMarkCapture002_Print();

END_PROGRAM

PROGRAM _EXIT
	(* Insert code here *)

END_PROGRAM
```

### Program Logical/SOURCE/VisCtrl/VisCtrl (IEC)

#### Main.st - Init, cyclic, exit code
```iecst
PROGRAM _INIT
	gPrintMarkHMI.Para.beltJogSpeed := K_BELT_JOG_INIT;
	gPrintMarkHMI.Para.cutterJogSpeed := K_CUTTER_JOG_INIT;
END_PROGRAM

PROGRAM _CYCLIC

	//Manual commands mapping for Belt conveyor axis
	gAx_BeltConveyor.In.Power := gPrintMarkHMI.Cmd.bBeltPowerOn;
	gAx_BeltConveyor.In.ErrorReset := gPrintMarkHMI.Cmd.bBeltErrorReset;
	IF(gAx_BeltConveyor.Out.IsHomed = TRUE)THEN
		gPrintMarkHMI.Cmd.bBeltHome := FALSE;
	END_IF;

	//Manual commands mapping for Cutter conveyor axis
	gAx_Cutter.In.Power := gPrintMarkHMI.Cmd.bCutterPowerOn;
	gAx_Cutter.In.ErrorReset := gPrintMarkHMI.Cmd.bCutterErrorReset;
	IF((gAx_Cutter.Out.IsHomed = TRUE) AND (gAx_Cutter.Out.Position = K_ZERO))THEN
		gPrintMarkHMI.Cmd.bCutterHome := FALSE;
	END_IF;

	//Animation;

END_PROGRAM

PROGRAM _EXIT
	(* Insert code here *)

END_PROGRAM
```

#### Types.typ - Local data types
```iecst
TYPE
	enAnimationSteps :
		(
		ZERO,
		FORTY_FIVE,
		NINETY,
		ONE_THIRTY_FIVE,
		THREE_SIXTY
		);
END_TYPE
```

#### Variables.var - Local variables
```iecst
(*Constants*)
VAR CONSTANT
	K_ZERO : USINT := 0; (*Constant zero value*)
	K_CUTTER_JOG_INIT : REAL := 100; (*Init value for cutter jog speed*)
	K_BELT_JOG_INIT : REAL := 100; (*Init value for belt jog speed*)
END_VAR
(*Enumeration variable*)
VAR
	enAnimation : enAnimationSteps;
END_VAR
```

#### Animation.st
```iecst
ACTION Animation:
	CASE enAnimation OF
		ZERO:
			gPrintMarkHMI.Para.beltAnimationString := '[{"select":"#svg1","spin":[45,0,0]}]';
			enAnimation := FORTY_FIVE;

		FORTY_FIVE:
				gPrintMarkHMI.Para.beltAnimationString := '[{"select":"#svg1","spin":[45,0,0]}]';
			enAnimation := NINETY;
		NINETY:
			gPrintMarkHMI.Para.beltAnimationString := '[{"select":"#svg1","spin":[45,0,0]}]';

			enAnimation := ONE_THIRTY_FIVE;
		ONE_THIRTY_FIVE:
				gPrintMarkHMI.Para.beltAnimationString  := '[{"select":"#svg1","spin":[45,0,0]}]';
		enAnimation := THREE_SIXTY;

		THREE_SIXTY:
				gPrintMarkHMI.Para.beltAnimationString := '[{"select":"#svg1","spin":[45,0,0]}]';
			enAnimation := ZERO;

	END_CASE;

END_ACTION
```

#### BeltAnime.st - not listed in the package file held
```iecst
ACTION BeltAnime:

	//Logic for belt animation
	IF(beltAnimation <= K_ANIMATION_LIMIT)THEN
		beltAnimation := beltAnimation + 1;
	ELSE
		beltAnimation := K_ZERO;
	END_IF;

END_ACTION
```

#### CutAnime.st - not listed in the package file held
```iecst
ACTION CutAnime:

	//Logic for cutter animation
	IF(cutterAnimation >= (-(K_ANIMATION_LIMIT)))THEN
		cutterAnimation := cutterAnimation - 1;
	ELSE
		cutterAnimation := K_ZERO;
	END_IF;

END_ACTION
```

### VisCtrl.typ
```iecst
(*HMI Structure for machine control*)

TYPE
	PrintCmdHMI_Typ : 	STRUCT
		bStart : BOOL; (*Start command via HMI*)
		bStop : BOOL; (*Start command via HMI*)
		bBeltJogPositive : BOOL; (*Belt Jog Positive command via HMI*)
		bBeltJogNegative : BOOL; (*Belt Jog Negative command via HMI*)
		bCutterJogPositive : BOOL; (*Cutter Jog Positive command via HMI*)
		bCutterJogNegative : BOOL; (*Cutter Jog Negative command via HMI*)
		bBeltPowerOn : BOOL; (*Belt conveyor axis power on*)
		bCutterPowerOn : BOOL; (*Cutter axis power on*)
		bBeltHome : BOOL; (*Belt axis home command*)
		bCutterHome : BOOL; (*Cutter axis home command*)
		bBeltErrorReset : BOOL; (*Belt conveyor axis error reset command*)
		bCutterErrorReset : BOOL; (*Cutter axis error reset command*)
	END_STRUCT;
	PrintParaHMI_Typ : 	STRUCT
		beltJogSpeed : REAL; (*Jog velocity for belt conveyor*)
		beltJogAcc : REAL; (*Jog acceleration for belt conveyor*)
		beltJogDecel : REAL; (*Jog deceleration for belt conveyor*)
		cutterJogSpeed : REAL; (*Jog velocity for cutter axis*)
		cutterJogAcc : REAL; (*Jog acceleration for cutter axis*)
		cutterJogDecel : REAL; (*Jog deceleration for cutter axis*)
		beltAnimationString : STRING[80]; (*Animation for belt conveyor*)
	END_STRUCT;
	PrintStatusHMI_Typ : 	STRUCT  (*Structure for showing the status of the machine*)
		New_Member : USINT;
	END_STRUCT;
	PrintInHMI_Typ : 	STRUCT  (*Structure for Inputs of the machine*)
		New_Member : USINT;
	END_STRUCT;
	PrintOutHMI_Typ : 	STRUCT  (*Structure for outputs of the machine*)
		New_Member : USINT;
	END_STRUCT;
	PrintIOHMI_Typ : 	STRUCT  (*Structure for IO's of the machine*)
		Input : PrintInHMI_Typ;
		Output : PrintOutHMI_Typ;
	END_STRUCT;
	PrintCtrHMIl_Typ : 	STRUCT  (*Structure of controlling the machine operation*)
		Cmd : PrintCmdHMI_Typ; (*Machine command type variable*)
		Status : PrintStatusHMI_Typ; (*Machine status type variable*)
		Para : PrintParaHMI_Typ; (*Machine parameter type variable*)
		IO : PrintIOHMI_Typ; (*Machine IO type variable*)
	END_STRUCT;
END_TYPE
```

### Program Logical/SOURCE/AlarmCtrl/AlarmCtrl

#### Variables.var
```iecst
(*Variables for MpAlarmxCore*)
VAR
	iFb_PrintMpAlarmXCore : MpAlarmXCore; (*Variable of MpAlarmxCore FB Type*)
	bAlarmXCoreReset : BOOL; (*Variable for reseting MpAlarmxCore FB*)
	iFb_PrintMpAlarmXListUI : MpAlarmXListUI; (*Variable for list of alarms*)
	printUIConnect : MpAlarmXListUIConnectType; (*Variable for list of alarms*)
END_VAR
```

#### Main.st
```iecst
(*|ŻŻŻŻŻŻŻŻŻŻŻŻŻŻŻŻŻŻŻŻŻŻŻŻŻŻŻŻŻŻŻŻŻŻŻŻŻŻŻŻŻŻŻŻŻŻŻŻŻŻŻŻŻŻŻŻŻŻŻŻŻŻŻŻŻŻŻŻŻŻŻŻŻŻ|*)
(*| Copyright      :- B&R Industrial Automation GmbH                         |*)
(*| Contact Person :-   kuma1p                                      		 |*)
(*|——————————————————————————————————————————————————————————————————————————|*)
(*| System       :-  Machine Name                                            |*)
(*| Task Name    :-  AlarmCtrl.st                                            |*)
(*| Auther Name  :-   kuma1p                                       			 |*)
(*| Created Date :-May 8, 2024/1:04 AM                                       |*)
(*| AS Version   :-  AS 4.12.2.93                                            |*)
(*|——————————————————————————————————————————————————————————————————————————|*)
(*| Description  :-  This task is for Alarm control                          |*)
(*|                                                                          |*)
(*|——————————————————————————————————————————————————————————————————————————|*)
(*| Version :-         V 0.0                      kuma1p                     |*)
(*|Changes Made :- Alarm Fb Added                                            |*)
(*|——————————————————————————————————————————————————————————————————————————|*)
PROGRAM _INIT

END_PROGRAM

PROGRAM _CYCLIC
	//Declaring MpAlarmXCore FB
	iFb_PrintMpAlarmXCore(MpLink := ADR(gMl_PrintAlarm) , Enable := TRUE , ErrorReset := bAlarmXCoreReset);
	//Declaring MpAlarmUIconnect FB
	iFb_PrintMpAlarmXListUI(MpLink := ADR(gMl_PrintAlarm) , Enable := TRUE ,UIConnect := ADR(printUIConnect) );

END_PROGRAM

PROGRAM _EXIT
//Exit Code
	iFb_PrintMpAlarmXCore(Enable := FALSE);
END_PROGRAM
```

### Program Logical/SOURCE/DataCtrl/DataCtrl

#### Variables.var
```iecst
(*Variable of MpDataRecorder type*)
VAR
	iFb_PrintMpDataRecorder : MpDataRecorder; (*Variable of MpDataRecorder type*)
	iFb_AvgMpDataRegPar : MpDataRegPar; (*VAriable of MpDataRegPar type*)
END_VAR
```

#### Main.st
```iecst
(*|ŻŻŻŻŻŻŻŻŻŻŻŻŻŻŻŻŻŻŻŻŻŻŻŻŻŻŻŻŻŻŻŻŻŻŻŻŻŻŻŻŻŻŻŻŻŻŻŻŻŻŻŻŻŻŻŻŻŻŻŻŻŻŻŻŻŻŻŻŻŻŻŻŻŻ|*)
(*| Copyright      :- B&R Industrial Automation GmbH                         |*)
(*| Contact Person :-   kuma1p                                      		 |*)
(*|——————————————————————————————————————————————————————————————————————————|*)
(*| System       :-  Machine Name                                            |*)
(*| Task Name    :-  DataCtrl.st                                             |*)
(*| Auther Name  :-   kuma1p                                       			 |*)
(*| Created Date :-May 8, 2024/1:04 AM                                       |*)
(*| AS Version   :-  AS 4.12.2.93                                            |*)
(*|——————————————————————————————————————————————————————————————————————————|*)
(*| Description  :-  This task is for Data control                           |*)
(*|                                                                          |*)
(*|——————————————————————————————————————————————————————————————————————————|*)
(*| Version :-         V 0.0                      kuma1p                     |*)
(*|Changes Made :-    Mp Data recorder fb added                              |*)
(*|——————————————————————————————————————————————————————————————————————————|*)
PROGRAM _INIT

END_PROGRAM

PROGRAM _CYCLIC
	//Calling MpData FB
	iFb_PrintMpDataRecorder(MpLink := ADR(gMl_PrintDataRecorder) , Enable := TRUE ,DeviceName := ADR('Print') , SamplingTime := T#1s, RecordMode := 2);
	//Caling MpDataRegPar for recording
	//Recording Processing time
	iFb_AvgMpDataRegPar(MpLink := ADR(gMl_PrintDataRecorder), Enable := TRUE ,PVName := ADR('gPrintMarkHMI.Para.avgPmDistance'));
	IF(gAx_CutterCam.Out.InSync = TRUE)THEN
		iFb_PrintMpDataRecorder.Record := TRUE;
	ELSE
		iFb_PrintMpDataRecorder.Record := FALSE;
	END_IF;

END_PROGRAM

PROGRAM _EXIT
	//Exit code
	iFb_PrintMpDataRecorder(Enable := FALSE);
	iFb_AvgMpDataRegPar(Enable := FALSE);
END_PROGRAM
```

### Program Logical/SOURCE/PackML/PackML (IEC)

#### Main.st - Init, cyclic, exit code
```iecst
(*|ŻŻŻŻŻŻŻŻŻŻŻŻŻŻŻŻŻŻŻŻŻŻŻŻŻŻŻŻŻŻŻŻŻŻŻŻŻŻŻŻŻŻŻŻŻŻŻŻŻŻŻŻŻŻŻŻŻŻŻŻŻŻŻŻŻŻŻŻŻŻŻŻŻŻ|*)
(*| Copyright      :- B&R Industrial Automation GmbH                         |*)
(*| Contact Person :-   kuma1p                                      		 |*)
(*|——————————————————————————————————————————————————————————————————————————|*)
(*| System       :-  Machine Name                                            |*)
(*| Task Name    :-  PackML.st                                               |*)
(*| Auther Name  :-   kuma1p                                       			 |*)
(*| Created Date :-May 8, 2024/1:04 AM                                       |*)
(*| AS Version   :-  AS 4.12.2.93                                            |*)
(*|——————————————————————————————————————————————————————————————————————————|*)
(*| Description  :-  This task is for PackMl Control                         |*)
(*|                                                                          |*)
(*|——————————————————————————————————————————————————————————————————————————|*)
(*| Version :-         V 0.0                      kuma1p                     |*)
(*|Changes Made :-     Pack ML fb added                                      |*)
(*|——————————————————————————————————————————————————————————————————————————|*)
PROGRAM _INIT

END_PROGRAM

PROGRAM _CYCLIC
	//Callig PackML Actions
	Core;
	Mode;

END_PROGRAM

PROGRAM _EXIT

END_PROGRAM
```

#### Variables.var - Local variables
```iecst
(*Variables of PackML Type*)
VAR
	iFb_MpPackMLModeAuto : MpPackMLMode; (*Variable for MpPackMLCore type*)
	iFb_MpPackMLModeManual : MpPackMLMode; (*Variable for MpPackMLMode type*)
	iFb_MpPackMLCorePrint : MpPackMLCore; (*Variable for MpPackMLMode type*)
END_VAR
```

#### Core.st - Pack ML core fb 
```iecst
ACTION Core:

	//Calling PackMLCore FB
	iFb_MpPackMLCorePrint(MpLink := ADR(gMl_PrintPackML) , Enable := TRUE);

END_ACTION
```

#### Mode.st - Pack ML Mode FB
```iecst
ACTION Mode:

	//Calling PackMLMode FB
	iFb_MpPackMLModeAuto(MpLink := ADR(gMl_PrintPackML) , Enable := TRUE ,  ModeID := 1 , Activate := TRUE);
	iFb_MpPackMLModeManual(MpLink := ADR(gMl_PrintPackML) , Enable := TRUE ,  ModeID := 2 , Activate := TRUE);

END_ACTION
```

- Visualisation Logical/mappView (not shown)

Listed in the project but not available here: Logical/acp10etxen, Logical/SOURCE/PackML/PackML/Types.typ
